  MoveL 5905 to (-69.95, 17.86, -237.76) mm, rotated rx -9.61 ry -16.54 rz -54.03 deg; joints [-14.429, -59.988, 109.983, 192.875, 34.389, -113.768, -415]
  MoveL 5906 to (-68.96, 18.06, -237.77) mm, rotated rx -9.61 ry -16.54 rz -54.03 deg; joints [-14.434, -59.99, 110.053, 192.844, 34.456, -113.734, -415]
  MoveL 5907 to (-67.92, 18.24, -237.77) mm, rotated rx -9.61 ry -16.54 rz -54.03 deg; joints [-14.44, -59.993, 110.127, 192.812, 34.524, -113.701, -415]
  MoveL 5908 to (-67.43, 18.33, -237.77) mm, rotated rx -9.61 ry -16.54 rz -54.03 deg; joints [-14.443, -59.994, 110.162, 192.796, 34.557, -113.684, -415]
  MoveL 5909 to (-66.78, 18.46, -237.8) mm, rotated rx -9.61 ry -16.54 rz -54.03 deg; joints [-14.447, -59.995, 110.208, 192.774, 34.6, -113.662, -415]
  MoveL 5910 to (-66.2, 18.59, -237.86) mm, rotated rx -9.61 ry -16.54 rz -54.03 deg; joints [-14.452, -59.994, 110.248, 192.753, 34.639, -113.64, -415]
  MoveL 5911 to (-65.71, 18.72, -237.93) mm, rotated rx -9.61 ry -16.54 rz -54.03 deg; joints [-14.457, -59.992, 110.28, 192.733, 34.671, -113.622, -415]
  MoveL 5912 to (-65.26, 18.83, -237.99) mm, rotated rx -9.61 ry -16.54 rz -54.03 deg; joints [-14.462, -59.99, 110.31, 192.716, 34.701, -113.605, -415]
  MoveL 5913 to (-64.81, 18.93, -238.02) mm, rotated rx -9.61 ry -16.54 rz -54.03 deg; joints [-14.465, -59.99, 110.341, 192.7, 34.732, -113.589, -415]
  MoveL 5914 to (-63.26, 19.2, -238.02) mm, rotated rx -9.61 ry -16.54 rz -54.03 deg; joints [-14.473, -59.994, 110.452, 192.653, 34.834, -113.539, -415]
  MoveL 5915 to (-62.77, 19.31, -238.03) mm, rotated rx -9.61 ry -16.54 rz -54.03 deg; joints [-14.476, -59.994, 110.486, 192.637, 34.867, -113.522, -415]
  MoveL 5916 to (-62.35, 19.42, -238.06) mm, rotated rx -9.61 ry -16.54 rz -54.03 deg; joints [-14.479, -59.992, 110.514, 192.622, 34.896, -113.507, -415]
  MoveL 5917 to (-61.98, 19.56, -238.11) mm, rotated rx -9.61 ry -16.54 rz -54.03 deg; joints [-14.483, -59.988, 110.537, 192.608, 34.922, -113.494, -415]
  MoveL 5918 to (-61.72, 19.71, -238.17) mm, rotated rx -9.61 ry -16.54 rz -54.03 deg; joints [-14.486, -59.981, 110.549, 192.596, 34.941, -113.482, -415]
  MoveL 5919 to (-61.52, 19.89, -238.24) mm, rotated rx -9.61 ry -16.54 rz -54.03 deg; joints [-14.49, -59.971, 110.558, 192.585, 34.958, -113.472, -415]
  MoveL 5920 to (-63.02, 19.39, -239.05) mm, rotated rx -9.61 ry -16.54 rz -54.03 deg; joints [-14.515, -59.976, 110.447, 192.579, 34.842, -113.488, -415]
  MoveL 5921 to (-61.72, 20.58, -239.45) mm, rotated rx -9.61 ry -16.54 rz -54.03 deg; joints [-14.534, -59.912, 110.497, 192.512, 34.95, -113.424, -415]
  MoveL 5922 to (-60.36, 21.87, -239.71) mm, rotated rx -9.61 ry -16.54 rz -54.03 deg; joints [-14.548, -59.843, 110.549, 192.452, 35.066, -113.364, -415]
  MoveL 5923 to (-58.92, 23.27, -239.9) mm, rotated rx -9.61 ry -16.54 rz -54.03 deg; joints [-14.558, -59.769, 110.603, 192.396, 35.191, -113.305, -415]
  MoveL 5924 to (-57.4, 24.77, -240.09) mm, rotated rx -9.61 ry -16.54 rz -54.03 deg; joints [-14.569, -59.688, 110.659, 192.336, 35.323, -113.243, -415]
  MoveL 5925 to (-55.87, 26.25, -240.18) mm, rotated rx -9.61 ry -16.54 rz -54.03 deg; joints [-14.576, -59.609, 110.718, 192.283, 35.457, -113.184, -415]
  MoveL 5926 to (-54.34, 27.74, -240.28) mm, rotated rx -9.61 ry -16.54 rz -54.03 deg; joints [-14.583, -59.529, 110.777, 192.231, 35.591, -113.126, -415]
  MoveL 5927 to (-52.81, 29.23, -240.48) mm, rotated rx -9.61 ry -16.54 rz -54.03 deg; joints [-14.594, -59.448, 110.833, 192.172, 35.723, -113.065, -415]
  MoveL 5928 to (-51.28, 30.71, -240.58) mm, rotated rx -9.61 ry -16.54 rz -54.03 deg; joints [-14.601, -59.369, 110.891, 192.12, 35.858, -113.008, -415]
  MoveL 5929 to (-49.74, 32.19, -240.68) mm, rotated rx -9.61 ry -16.54 rz -54.03 deg; joints [-14.609, -59.289, 110.949, 192.068, 35.991, -112.951, -415]
  MoveL 5930 to (-48.2, 33.67, -240.88) mm, rotated rx -9.61 ry -16.54 rz -54.03 deg; joints [-14.62, -59.207, 111.005, 192.011, 36.124, -112.891, -415]
  MoveL 5931 to (-45.12, 36.63, -241.08) mm, rotated rx -9.61 ry -16.54 rz -54.03 deg; joints [-14.635, -59.046, 111.12, 191.909, 36.392, -112.779, -415]
  MoveL 5932 to (-43.83, 37.86, -241.29) mm, rotated rx -9.61 ry -16.54 rz -54.03 deg; joints [-14.646, -58.978, 111.167, 191.859, 36.504, -112.728, -415]
  MoveL 5933 to (-42.44, 39.25, -241.36) mm, rotated rx -9.61 ry -16.54 rz -54.03 deg; joints [-14.652, -58.901, 111.216, 191.815, 36.626, -112.679, -415]
  MoveL 5934 to (-41.02, 40.74, -241.37) mm, rotated rx -9.61 ry -16.54 rz -54.03 deg; joints [-14.655, -58.818, 111.264, 191.775, 36.754, -112.631, -415]
  MoveL 5935 to (-39.08, 42.58, -241.48) mm, rotated rx -9.61 ry -16.54 rz -54.03 deg; joints [-14.663, -58.717, 111.335, 191.714, 36.922, -112.563, -415]
  MoveL 5936 to (-37.13, 44.27, -241.58) mm, rotated rx -9.61 ry -16.54 rz -54.03 deg; joints [-14.672, -58.625, 111.413, 191.655, 37.087, -112.498, -415]
  MoveL 5937 to (-35.51, 45.76, -241.67) mm, rotated rx -9.61 ry -16.54 rz -54.03 deg; joints [-14.68, -58.542, 111.475, 191.604, 37.227, -112.442, -415]
  MoveL 5938 to (-34.01, 47.16, -241.84) mm, rotated rx -9.61 ry -16.54 rz -54.03 deg; joints [-14.69, -58.464, 111.528, 191.553, 37.355, -112.389, -415]
  MoveL 5939 to (-32.61, 48.45, -242.13) mm, rotated rx -9.61 ry -16.54 rz -54.03 deg; joints [-14.704, -58.39, 111.577, 191.498, 37.473, -112.334, -415]
  MoveL 5940 to (-31.22, 49.73, -242.41) mm, rotated rx -9.61 ry -16.54 rz -54.03 deg; joints [-14.719, -58.316, 111.625, 191.444, 37.591, -112.28, -415]
  MoveL 5941 to (-29.81, 50.98, -242.71) mm, rotated rx -9.61 ry -16.54 rz -54.03 deg; joints [-14.734, -58.245, 111.675, 191.389, 37.708, -112.226, -415]
  MoveL 5942 to (-28.34, 52.33, -242.86) mm, rotated rx -9.61 ry -16.54 rz -54.03 deg; joints [-14.744, -58.169, 111.728, 191.341, 37.833, -112.176, -415]
  MoveL 5943 to (-27.69, 52.32, -243.48) mm, rotated rx -9.61 ry -16.54 rz -54.03 deg; joints [-14.773, -58.171, 111.768, 191.286, 37.867, -112.136, -415]
  MoveL 5944 to (-27.8, 52.02, -243.79) mm, rotated rx -9.61 ry -16.54 rz -54.03 deg; joints [-14.786, -58.188, 111.767, 191.271, 37.849, -112.129, -415]
  MoveL 5945 to (-27.77, 51.98, -243.98) mm, rotated rx -9.61 ry -16.54 rz -54.03 deg; joints [-14.794, -58.189, 111.768, 191.258, 37.847, -112.122, -415]
  MoveL 5946 to (-27.63, 52.19, -244.08) mm, rotated rx -9.61 ry -16.54 rz -54.03 deg; joints [-14.798, -58.176, 111.768, 191.249, 37.86, -112.114, -415]
  MoveL 5947 to (-27.45, 52.6, -244.1) mm, rotated rx -9.61 ry -16.54 rz -54.03 deg; joints [-14.798, -58.15, 111.764, 191.243, 37.882, -112.107, -415]
  MoveL 5948 to (-27.29, 53.06, -244.1) mm, rotated rx -9.61 ry -16.54 rz -54.03 deg; joints [-14.798, -58.12, 111.757, 191.238, 37.904, -112.1, -415]
  MoveL 5949 to (-27.08, 54.01, -244.14) mm, rotated rx -9.61 ry -16.54 rz -54.03 deg; joints [-14.796, -58.058, 111.733, 191.231, 37.941, -112.089, -415]
  MoveL 5950 to (-26.74, 55.55, -244.14) mm, rotated rx -9.61 ry -16.54 rz -54.03 deg; joints [-14.792, -57.958, 111.694, 191.222, 38.002, -112.074, -415]
  MoveL 5951 to (-26.49, 56.5, -244.15) mm, rotated rx -9.61 ry -16.54 rz -54.03 deg; joints [-14.79, -57.896, 111.672, 191.215, 38.041, -112.063, -415]
  MoveL 5952 to (-26.27, 57.52, -244.15) mm, rotated rx -9.61 ry -16.54 rz -54.03 deg; joints [-14.788, -57.829, 111.646, 191.209, 38.081, -112.053, -415]
  MoveL 5953 to (-26.15, 58.02, -244.17) mm, rotated rx -9.61 ry -16.54 rz -54.03 deg; joints [-14.787, -57.796, 111.633, 191.205, 38.101, -112.047, -415]
  MoveL 5954 to (-26.04, 58.48, -244.2) mm, rotated rx -9.61 ry -16.54 rz -54.03 deg; joints [-14.787, -57.767, 111.622, 191.2, 38.12, -112.041, -415]
  MoveL 5955 to (-25.92, 58.9, -244.24) mm, rotated rx -9.61 ry -16.54 rz -54.03 deg; joints [-14.788, -57.739, 111.612, 191.194, 38.137, -112.035, -415]
  MoveL 5956 to (-25.81, 59.29, -244.31) mm, rotated rx -9.61 ry -16.54 rz -54.03 deg; joints [-14.789, -57.713, 111.604, 191.188, 38.153, -112.028, -415]
  MoveL 5957 to (-25.69, 59.69, -244.36) mm, rotated rx -9.61 ry -16.54 rz -54.03 deg; joints [-14.791, -57.687, 111.595, 191.182, 38.17, -112.021, -415]
  MoveL 5958 to (-25.57, 60.14, -244.39) mm, rotated rx -9.61 ry -16.54 rz -54.03 deg; joints [-14.791, -57.658, 111.584, 191.177, 38.188, -112.015, -415]
  MoveL 5959 to (-25.46, 60.6, -244.42) mm, rotated rx -9.61 ry -16.54 rz -54.03 deg; joints [-14.791, -57.627, 111.573, 191.172, 38.207, -112.009, -415]
  MoveL 5960 to (-25.34, 61.02, -244.46) mm, rotated rx -9.61 ry -16.54 rz -54.03 deg; joints [-14.792, -57.6, 111.563, 191.167, 38.225, -112.003, -415]
  MoveL 5961 to (-25.21, 61.41, -244.52) mm, rotated rx -9.61 ry -16.54 rz -54.03 deg; joints [-14.793, -57.575, 111.556, 191.16, 38.242, -111.996, -415]
  MoveL 5962 to (-25.09, 61.8, -244.57) mm, rotated rx -9.61 ry -16.54 rz -54.03 deg; joints [-14.794, -57.549, 111.547, 191.154, 38.259, -111.99, -415]
  MoveL 5963 to (-24.97, 62.22, -244.6) mm, rotated rx -9.61 ry -16.54 rz -54.03 deg; joints [-14.795, -57.521, 111.537, 191.149, 38.276, -111.984, -415]
  MoveL 5964 to (-24.86, 62.73, -244.6) mm, rotated rx -9.61 ry -16.54 rz -54.03 deg; joints [-14.793, -57.488, 111.524, 191.146, 38.296, -111.979, -415]
  MoveL 5965 to (-23.99, 65.52, -244.96) mm, rotated rx -9.61 ry -16.54 rz -54.03 deg; joints [-14.802, -57.306, 111.465, 191.103, 38.416, -111.933, -415]
  MoveL 5966 to (-23.41, 66.67, -245.4) mm, rotated rx -9.61 ry -16.54 rz -54.03 deg; joints [-14.818, -57.23, 111.452, 191.063, 38.476, -111.898, -415]
  MoveL 5967 to (-22.74, 67.66, -246.03) mm, rotated rx -9.61 ry -16.54 rz -54.03 deg; joints [-14.843, -57.164, 111.451, 191.009, 38.536, -111.855, -415]
  MoveL 5968 to (-21.11, 69.17, -247.81) mm, rotated rx -9.61 ry -16.54 rz -54.03 deg; joints [-14.918, -57.064, 111.48, 190.863, 38.655, -111.747, -415]
  MoveL 5969 to (-19.1, 70.04, -250.3) mm, rotated rx -9.61 ry -16.54 rz -54.03 deg; joints [-15.027, -57.003, 111.553, 190.666, 38.775, -111.607, -415]
  MoveL 5970 to (-17.3, 70.14, -252.79) mm, rotated rx -9.61 ry -16.54 rz -54.03 deg; joints [-15.138, -56.991, 111.643, 190.475, 38.863, -111.477, -415]
  MoveL 5971 to (-16.71, 69.87, -253.77) mm, rotated rx -9.61 ry -16.54 rz -54.03 deg; joints [-15.182, -57.008, 111.684, 190.402, 38.882, -111.43, -415]
  MoveL 5972 to (-16.31, 69.36, -254.58) mm, rotated rx -9.61 ry -16.54 rz -54.03 deg; joints [-15.218, -57.038, 111.722, 190.345, 38.886, -111.395, -415]
  MoveL 5973 to (-16.19, 69.03, -254.91) mm, rotated rx -9.61 ry -16.54 rz -54.03 deg; joints [-15.234, -57.059, 111.74, 190.321, 38.881, -111.382, -415]
  MoveL 5974 to (-16.12, 68.64, -255.2) mm, rotated rx -9.61 ry -16.54 rz -54.03 deg; joints [-15.248, -57.084, 111.757, 190.302, 38.873, -111.371, -415]
  MoveL 5975 to (-16.13, 67.69, -255.64) mm, rotated rx -9.61 ry -16.54 rz -54.03 deg; joints [-15.269, -57.144, 111.79, 190.275, 38.844, -111.359, -415]
  MoveL 5976 to (-16.34, 66.52, -255.91) mm, rotated rx -9.61 ry -16.54 rz -54.03 deg; joints [-15.284, -57.219, 111.82, 190.263, 38.798, -111.359, -415]
  MoveL 5977 to (-16.76, 65.13, -256) mm, rotated rx -9.61 ry -16.54 rz -54.03 deg; joints [-15.291, -57.308, 111.847, 190.267, 38.736, -111.37, -415]
  MoveL 5978 to (-17.61, 62.66, -256) mm, rotated rx -9.61 ry -16.54 rz -54.03 deg; joints [-15.296, -57.468, 111.89, 190.285, 38.621, -111.399, -415]
  MoveL 5979 to (-17.76, 62.25, -255.97) mm, rotated rx -9.61 ry -16.54 rz -54.03 deg; joints [-15.295, -57.494, 111.896, 190.29, 38.601, -111.405, -415]
  MoveL 5980 to (-17.92, 61.87, -255.92) mm, rotated rx -9.61 ry -16.54 rz -54.03 deg; joints [-15.294, -57.518, 111.901, 190.296, 38.582, -111.412, -415]
  MoveL 5981 to (-18.08, 61.52, -255.85) mm, rotated rx -9.61 ry -16.54 rz -54.03 deg; joints [-15.292, -57.541, 111.906, 190.304, 38.564, -111.42, -415]
  MoveL 5982 to (-18.24, 61.12, -255.8) mm, rotated rx -9.61 ry -16.54 rz -54.03 deg; joints [-15.29, -57.567, 111.911, 190.311, 38.544, -111.427, -415]
  MoveL 5983 to (-18.42, 60.66, -255.76) mm, rotated rx -9.61 ry -16.54 rz -54.03 deg; joints [-15.29, -57.597, 111.918, 190.317, 38.522, -111.434, -415]
  MoveL 5984 to (-18.62, 60.17, -255.71) mm, rotated rx -9.61 ry -16.54 rz -54.03 deg; joints [-15.288, -57.629, 111.925, 190.325, 38.497, -111.442, -415]
  MoveL 5985 to (-18.81, 59.66, -255.69) mm, rotated rx -9.61 ry -16.54 rz -54.03 deg; joints [-15.288, -57.661, 111.933, 190.33, 38.473, -111.449, -415]
  MoveL 5986 to (-19.01, 59.05, -255.7) mm, rotated rx -9.61 ry -16.54 rz -54.03 deg; joints [-15.29, -57.7, 111.943, 190.333, 38.444, -111.456, -415]
  MoveL 5987 to (-19.27, 58.22, -255.77) mm, rotated rx -9.61 ry -16.54 rz -54.03 deg; joints [-15.295, -57.754, 111.958, 190.335, 38.406, -111.463, -415]
  MoveL 5988 to (-19.44, 57.72, -255.77) mm, rotated rx -9.61 ry -16.54 rz -54.03 deg; joints [-15.296, -57.785, 111.966, 190.339, 38.383, -111.468, -415]
  MoveL 5989 to (-19.6, 57.25, -255.76) mm, rotated rx -9.61 ry -16.54 rz -54.03 deg; joints [-15.297, -57.816, 111.974, 190.343, 38.361, -111.474, -415]
  MoveL 5990 to (-19.76, 56.82, -255.74) mm, rotated rx -9.61 ry -16.54 rz -54.03 deg; joints [-15.297, -57.844, 111.981, 190.348, 38.34, -111.481, -415]
  MoveL 5991 to (-19.92, 56.43, -255.69) mm, rotated rx -9.61 ry -16.54 rz -54.03 deg; joints [-15.295, -57.869, 111.985, 190.354, 38.32, -111.488, -415]
  MoveL 5992 to (-20.09, 56.07, -255.63) mm, rotated rx -9.61 ry -16.54 rz -54.03 deg; joints [-15.293, -57.892, 111.989, 190.362, 38.301, -111.495, -415]
  MoveL 5993 to (-20.31, 55.71, -255.58) mm, rotated rx -9.61 ry -16.54 rz -54.03 deg; joints [-15.291, -57.914, 111.988, 190.37, 38.279, -111.504, -415]
  MoveL 5994 to (-20.56, 55.39, -255.52) mm, rotated rx -9.61 ry -16.54 rz -54.03 deg; joints [-15.289, -57.935, 111.984, 190.379, 38.255, -111.513, -415]
  MoveL 5995 to (-20.74, 55.25, -255.36) mm, rotated rx -9.61 ry -16.54 rz -54.03 deg; joints [-15.282, -57.943, 111.979, 190.394, 38.242, -111.524, -415]
  MoveL 5996 to (-20.74, 55.36, -255.05) mm, rotated rx -9.61 ry -16.54 rz -54.03 deg; joints [-15.269, -57.939, 111.979, 190.413, 38.248, -111.534, -415]
  MoveL 5997 to (-20.54, 55.75, -254.56) mm, rotated rx -9.61 ry -16.54 rz -54.03 deg; joints [-15.249, -57.919, 111.987, 190.437, 38.277, -111.545, -415]
  MoveL 5998 to (-21.22, 55.18, -253.71) mm, rotated rx -9.61 ry -16.54 rz -54.03 deg; joints [-15.212, -57.957, 111.973, 190.505, 38.229, -111.594, -415]
  MoveL 5999 to (-24.62, 52.6, -253.71) mm, rotated rx -9.61 ry -16.54 rz -54.03 deg; joints [-15.202, -58.097, 111.825, 190.589, 37.948, -111.689, -415]
  MoveL 6000 to (-26.22, 51.39, -253.64) mm, rotated rx -9.61 ry -16.54 rz -54.03 deg; joints [-15.194, -58.162, 111.756, 190.632, 37.817, -111.737, -415]
  MoveL 6001 to (-27.81, 50.2, -253.49) mm, rotated rx -9.61 ry -16.54 rz -54.03 deg; joints [-15.183, -58.227, 111.688, 190.681, 37.687, -111.788, -415]
  MoveL 6002 to (-29.65, 48.83, -253.3) mm, rotated rx -9.61 ry -16.54 rz -54.03 deg; joints [-15.17, -58.301, 111.609, 190.739, 37.538, -111.847, -415]
  MoveL 6003 to (-31.39, 47.53, -253.08) mm, rotated rx -9.61 ry -16.54 rz -54.03 deg; joints [-15.156, -58.371, 111.534, 190.797, 37.397, -111.905, -415]
  MoveL 6004 to (-33.13, 46.22, -252.98) mm, rotated rx -9.61 ry -16.54 rz -54.03 deg; joints [-15.146, -58.441, 111.458, 190.848, 37.255, -111.96, -415]
  MoveL 6005 to (-34.83, 44.93, -252.98) mm, rotated rx -9.61 ry -16.54 rz -54.03 deg; joints [-15.141, -58.509, 111.382, 190.892, 37.114, -112.01, -415]
  MoveL 6006 to (-36.41, 43.72, -252.92) mm, rotated rx -9.61 ry -16.54 rz -54.03 deg; joints [-15.134, -58.572, 111.312, 190.937, 36.984, -112.059, -415]
  MoveL 6007 to (-37.9, 42.58, -252.8) mm, rotated rx -9.61 ry -16.54 rz -54.03 deg; joints [-15.124, -58.633, 111.247, 190.983, 36.862, -112.108, -415]
  MoveL 6008 to (-39.53, 41.35, -252.73) mm, rotated rx -9.61 ry -16.54 rz -54.03 deg; joints [-15.117, -58.697, 111.174, 191.03, 36.729, -112.159, -415]
  MoveL 6009 to (-41.22, 40.05, -252.55) mm, rotated rx -9.61 ry -16.54 rz -54.03 deg; joints [-15.104, -58.765, 111.1, 191.087, 36.591, -112.217, -415]
  MoveL 6010 to (-44.62, 37.46, -252.37) mm, rotated rx -9.61 ry -16.54 rz -54.03 deg; joints [-15.087, -58.899, 110.948, 191.19, 36.312, -112.328, -415]
  MoveL 6011 to (-46.31, 36.16, -252.19) mm, rotated rx -9.61 ry -16.54 rz -54.03 deg; joints [-15.074, -58.967, 110.873, 191.247, 36.174, -112.387, -415]
  MoveL 6012 to (-48, 34.85, -252.01) mm, rotated rx -9.61 ry -16.54 rz -54.03 deg; joints [-15.062, -59.034, 110.799, 191.305, 36.036, -112.447, -415]
  MoveL 6013 to (-49.7, 33.56, -252.01) mm, rotated rx -9.61 ry -16.54 rz -54.03 deg; joints [-15.057, -59.099, 110.72, 191.352, 35.896, -112.501, -415]
  MoveL 6014 to (-51.38, 32.25, -251.83) mm, rotated rx -9.61 ry -16.54 rz -54.03 deg; joints [-15.045, -59.166, 110.645, 191.411, 35.758, -112.561, -415]
  MoveL 6015 to (-53.06, 30.94, -251.66) mm, rotated rx -9.61 ry -16.54 rz -54.03 deg; joints [-15.033, -59.233, 110.57, 191.47, 35.62, -112.622, -415]
  MoveL 6016 to (-54.76, 29.65, -251.66) mm, rotated rx -9.61 ry -16.54 rz -54.03 deg; joints [-15.028, -59.297, 110.49, 191.518, 35.48, -112.677, -415]
  MoveL 6017 to (-56.27, 28.41, -251.46) mm, rotated rx -9.61 ry -16.54 rz -54.03 deg; joints [-15.016, -59.361, 110.425, 191.574, 35.355, -112.734, -415]
  MoveL 6018 to (-57.55, 27.27, -251.14) mm, rotated rx -9.61 ry -16.54 rz -54.03 deg; joints [-15, -59.422, 110.376, 191.632, 35.249, -112.789, -415]
  MoveL 6019 to (-58.64, 26.2, -250.68) mm, rotated rx -9.61 ry -16.54 rz -54.03 deg; joints [-14.979, -59.483, 110.341, 191.693, 35.158, -112.845, -415]
  MoveL 6020 to (-57.79, 26.63, -249.91) mm, rotated rx -9.61 ry -16.54 rz -54.03 deg; joints [-14.952, -59.473, 110.402, 191.718, 35.231, -112.849, -415]
  MoveL 6021 to (-58.15, 26.41, -249.9) mm, rotated rx -9.61 ry -16.54 rz -54.03 deg; joints [-14.95, -59.482, 110.383, 191.729, 35.204, -112.861, -415]
  MoveC 6022 to (-61.66, 25.91, -249.9) mm, rotated rx -9.61 ry -16.54 rz -54.03 deg; joints [-14.931, -59.467, 110.129, 191.83, 34.972, -112.967, -415] to (-65.21, 25.71, -249.9) mm, rotated rx -9.61 ry -16.54 rz -54.03 deg; joints [-14.91, -59.43, 109.859, 191.934, 34.747, -113.073, -415]
  MoveL 6023 to (-65.21, 25.71, -249.9) mm, rotated rx -9.61 ry -16.54 rz -54.03 deg; joints [-14.91, -59.43, 109.859, 191.934, 34.747, -113.073, -415]
  MoveL 6024 to (-65.68, 25.67, -249.88) mm, rotated rx -9.61 ry -16.54 rz -54.03 deg; joints [-14.907, -59.426, 109.825, 191.949, 34.717, -113.088, -415]
  MoveL 6025 to (-66.1, 25.62, -249.83) mm, rotated rx -9.61 ry -16.54 rz -54.03 deg; joints [-14.902, -59.425, 109.795, 191.964, 34.691, -113.103, -415]
  MoveL 6026 to (-66.5, 25.56, -249.77) mm, rotated rx -9.61 ry -16.54 rz -54.03 deg; joints [-14.898, -59.423, 109.767, 191.98, 34.665, -113.118, -415]
  MoveL 6027 to (-66.94, 25.51, -249.72) mm, rotated rx -9.61 ry -16.54 rz -54.03 deg; joints [-14.893, -59.421, 109.735, 191.996, 34.637, -113.133, -415]
  MoveL 6028 to (-67.41, 25.46, -249.7) mm, rotated rx -9.61 ry -16.54 rz -54.03 deg; joints [-14.89, -59.417, 109.7, 192.012, 34.607, -113.149, -415]
  MoveL 6029 to (-67.93, 25.43, -249.68) mm, rotated rx -9.61 ry -16.54 rz -54.03 deg; joints [-14.886, -59.412, 109.662, 192.028, 34.575, -113.165, -415]
  MoveL 6030 to (-68.97, 25.36, -249.68) mm, rotated rx -9.61 ry -16.54 rz -54.03 deg; joints [-14.88, -59.401, 109.582, 192.059, 34.508, -113.197, -415]
  MoveL 6031 to (-70.43, 25.33, -249.77) mm, rotated rx -9.61 ry -16.54 rz -54.03 deg; joints [-14.875, -59.381, 109.467, 192.096, 34.416, -113.238, -415]
  MoveL 6032 to (-71.62, 25.43, -250.05) mm, rotated rx -9.61 ry -16.54 rz -54.03 deg; joints [-14.878, -59.355, 109.365, 192.114, 34.342, -113.262, -415]
  MoveL 6033 to (-72.56, 25.67, -250.5) mm, rotated rx -9.61 ry -16.54 rz -54.03 deg; joints [-14.89, -59.322, 109.275, 192.112, 34.285, -113.271, -415]
  MoveL 6034 to (-73.24, 26.03, -251.14) mm, rotated rx -9.61 ry -16.54 rz -54.03 deg; joints [-14.91, -59.282, 109.197, 192.09, 34.244, -113.263, -415]
  MoveL 6035 to (-73.67, 26.52, -251.97) mm, rotated rx -9.61 ry -16.54 rz -54.03 deg; joints [-14.938, -59.236, 109.131, 192.049, 34.221, -113.239, -415]
  MoveL 6036 to (-73.83, 27.14, -252.97) mm, rotated rx -9.61 ry -16.54 rz -54.03 deg; joints [-14.974, -59.183, 109.077, 191.988, 34.215, -113.198, -415]
  MoveL 6037 to (-73.39, 28.77, -255.53) mm, rotated rx -9.61 ry -16.54 rz -54.03 deg; joints [-15.071, -59.059, 109.007, 191.807, 34.255, -113.07, -415]
  MoveL 6038 to (-72.15, 30.4, -258.09) mm, rotated rx -9.61 ry -16.54 rz -54.03 deg; joints [-15.173, -58.946, 108.997, 191.604, 34.343, -112.918, -415]
  MoveL 6039 to (-71.32, 31.03, -259.1) mm, rotated rx -9.61 ry -16.54 rz -54.03 deg; joints [-15.215, -58.907, 109.021, 191.515, 34.399, -112.849, -415]
  MoveL 6040 to (-70.36, 31.53, -259.92) mm, rotated rx -9.61 ry -16.54 rz -54.03 deg; joints [-15.252, -58.881, 109.063, 191.434, 34.462, -112.785, -415]
  MoveL 6041 to (-69.26, 31.9, -260.56) mm, rotated rx -9.61 ry -16.54 rz -54.03 deg; joints [-15.282, -58.866, 109.124, 191.36, 34.532, -112.724, -415]
  MoveL 6042 to (-68.01, 32.14, -261.02) mm, rotated rx -9.61 ry -16.54 rz -54.03 deg; joints [-15.307, -58.864, 109.204, 191.295, 34.61, -112.669, -415]
  MoveL 6043 to (-65.12, 32.24, -261.38) mm, rotated rx -9.61 ry -16.54 rz -54.03 deg; joints [-15.339, -58.894, 109.421, 191.189, 34.788, -112.57, -415]
  MoveL 6044 to (-64.07, 32.19, -261.38) mm, rotated rx -9.61 ry -16.54 rz -54.03 deg; joints [-15.346, -58.912, 109.505, 191.159, 34.852, -112.54, -415]
  MoveL 6045 to (-63.55, 32.17, -261.39) mm, rotated rx -9.61 ry -16.54 rz -54.03 deg; joints [-15.35, -58.921, 109.546, 191.144, 34.884, -112.525, -415]
  MoveL 6046 to (-63.07, 32.16, -261.41) mm, rotated rx -9.61 ry -16.54 rz -54.03 deg; joints [-15.354, -58.928, 109.583, 191.129, 34.913, -112.51, -415]
  MoveL 6047 to (-62.65, 32.17, -261.46) mm, rotated rx -9.61 ry -16.54 rz -54.03 deg; joints [-15.358, -58.933, 109.616, 191.114, 34.939, -112.496, -415]
  MoveL 6048 to (-62.25, 32.18, -261.52) mm, rotated rx -9.61 ry -16.54 rz -54.03 deg; joints [-15.363, -58.937, 109.646, 191.099, 34.963, -112.483, -415]
  MoveL 6049 to (-61.83, 32.18, -261.56) mm, rotated rx -9.61 ry -16.54 rz -54.03 deg; joints [-15.367, -58.942, 109.677, 191.084, 34.989, -112.469, -415]
  MoveL 6050 to (-61.36, 32.17, -261.59) mm, rotated rx -9.61 ry -16.54 rz -54.03 deg; joints [-15.371, -58.949, 109.714, 191.07, 35.018, -112.455, -415]
  MoveL 6051 to (-60.86, 32.15, -261.59) mm, rotated rx -9.61 ry -16.54 rz -54.03 deg; joints [-15.375, -58.957, 109.753, 191.056, 35.048, -112.44, -415]
  MoveL 6052 to (-60.31, 32.12, -261.59) mm, rotated rx -9.61 ry -16.54 rz -54.03 deg; joints [-15.378, -58.967, 109.798, 191.041, 35.082, -112.425, -415]
  MoveL 6053 to (-59.78, 32.1, -261.59) mm, rotated rx -9.61 ry -16.54 rz -54.03 deg; joints [-15.382, -58.976, 109.84, 191.025, 35.114, -112.41, -415]
  MoveL 6054 to (-59.29, 32.09, -261.62) mm, rotated rx -9.61 ry -16.54 rz -54.03 deg; joints [-15.386, -58.983, 109.878, 191.01, 35.144, -112.395, -415]
  MoveL 6055 to (-58.81, 32.08, -261.66) mm, rotated rx -9.61 ry -16.54 rz -54.03 deg; joints [-15.391, -58.989, 109.914, 190.994, 35.173, -112.38, -415]
  MoveL 6056 to (-58.31, 32.1, -261.74) mm, rotated rx -9.61 ry -16.54 rz -54.03 deg; joints [-15.397, -58.995, 109.952, 190.975, 35.204, -112.363, -415]
  MoveL 6057 to (-57.7, 32.11, -261.8) mm, rotated rx -9.61 ry -16.54 rz -54.03 deg; joints [-15.403, -59.002, 109.997, 190.954, 35.241, -112.343, -415]
  MoveL 6058 to (-57.13, 32.09, -261.82) mm, rotated rx -9.61 ry -16.54 rz -54.03 deg; joints [-15.408, -59.01, 110.042, 190.937, 35.276, -112.327, -415]
  MoveL 6059 to (-56.61, 32.07, -261.82) mm, rotated rx -9.61 ry -16.54 rz -54.03 deg; joints [-15.411, -59.019, 110.084, 190.922, 35.308, -112.312, -415]
  MoveL 6060 to (-56.08, 32.04, -261.82) mm, rotated rx -9.61 ry -16.54 rz -54.03 deg; joints [-15.415, -59.027, 110.125, 190.908, 35.34, -112.298, -415]
  MoveL 6061 to (-55.42, 32.03, -261.83) mm, rotated rx -9.61 ry -16.54 rz -54.03 deg; joints [-15.419, -59.037, 110.177, 190.889, 35.381, -112.279, -415]
  MoveL 6062 to (-54.84, 32.04, -261.84) mm, rotated rx -9.61 ry -16.54 rz -54.03 deg; joints [-15.423, -59.044, 110.222, 190.873, 35.417, -112.262, -415]
  MoveL 6063 to (-54.33, 32.07, -261.85) mm, rotated rx -9.61 ry -16.54 rz -54.03 deg; joints [-15.427, -59.048, 110.259, 190.858, 35.449, -112.248, -415]
  MoveL 6064 to (-54, 32.15, -261.85) mm, rotated rx -9.61 ry -16.54 rz -54.03 deg; joints [-15.429, -59.048, 110.282, 190.849, 35.472, -112.238, -415]
  MoveL 6065 to (-53.75, 32.25, -261.85) mm, rotated rx -9.61 ry -16.54 rz -54.03 deg; joints [-15.43, -59.044, 110.298, 190.842, 35.491, -112.231, -415]
  MoveL 6066 to (-54.61, 31.88, -262.44) mm, rotated rx -9.61 ry -16.54 rz -54.03 deg; joints [-15.449, -59.052, 110.235, 190.828, 35.42, -112.233, -415]
  MoveL 6067 to (-53.63, 32.79, -262.97) mm, rotated rx -9.61 ry -16.54 rz -54.03 deg; joints [-15.473, -58.999, 110.266, 190.768, 35.499, -112.181, -415]
  MoveL 6068 to (-52.4, 33.75, -263.35) mm, rotated rx -9.61 ry -16.54 rz -54.03 deg; joints [-15.492, -58.948, 110.317, 190.71, 35.597, -112.128, -415]
  MoveL 6069 to (-50.87, 34.78, -263.61) mm, rotated rx -9.61 ry -16.54 rz -54.03 deg; joints [-15.507, -58.897, 110.389, 190.653, 35.716, -112.073, -415]
  MoveL 6070 to (-49.13, 35.87, -263.74) mm, rotated rx -9.61 ry -16.54 rz -54.03 deg; joints [-15.519, -58.846, 110.478, 190.598, 35.853, -112.017, -415]
  MoveL 6071 to (-47.33, 36.97, -263.83) mm, rotated rx -9.61 ry -16.54 rz -54.03 deg; joints [-15.529, -58.794, 110.57, 190.545, 35.993, -111.961, -415]
  MoveL 6072 to (-43.69, 39.18, -264.01) mm, rotated rx -9.61 ry -16.54 rz -54.03 deg; joints [-15.55, -58.69, 110.758, 190.438, 36.277, -111.849, -415]
  MoveL 6073 to (-41.87, 40.3, -264.19) mm, rotated rx -9.61 ry -16.54 rz -54.03 deg; joints [-15.564, -58.636, 110.849, 190.38, 36.419, -111.79, -415]
  MoveL 6074 to (-38.22, 42.51, -264.37) mm, rotated rx -9.61 ry -16.54 rz -54.03 deg; joints [-15.586, -58.53, 111.035, 190.275, 36.704, -111.681, -415]
  MoveL 6075 to (-36.39, 43.61, -264.55) mm, rotated rx -9.61 ry -16.54 rz -54.03 deg; joints [-15.6, -58.475, 111.126, 190.218, 36.845, -111.624, -415]
  MoveL 6076 to (-34.56, 44.71, -264.64) mm, rotated rx -9.61 ry -16.54 rz -54.03 deg; joints [-15.611, -58.422, 111.218, 190.166, 36.988, -111.57, -415]
  MoveL 6077 to (-32.86, 45.71, -264.86) mm, rotated rx -9.61 ry -16.54 rz -54.03 deg; joints [-15.626, -58.372, 111.303, 190.111, 37.119, -111.516, -415]
  MoveL 6078 to (-30.84, 46.93, -265) mm, rotated rx -9.61 ry -16.54 rz -54.03 deg; joints [-15.639, -58.311, 111.404, 190.052, 37.276, -111.456, -415]
  MoveL 6079 to (-28.64, 48.25, -265.12) mm, rotated rx -9.61 ry -16.54 rz -54.03 deg; joints [-15.653, -58.245, 111.513, 189.991, 37.447, -111.392, -415]
  MoveL 6080 to (-26.82, 49.35, -265.12) mm, rotated rx -9.61 ry -16.54 rz -54.03 deg; joints [-15.66, -58.191, 111.606, 189.947, 37.591, -111.344, -415]
  MoveL 6081 to (-25.07, 50.39, -265.2) mm, rotated rx -9.61 ry -16.54 rz -54.03 deg; joints [-15.67, -58.139, 111.693, 189.9, 37.728, -111.295, -415]
  MoveL 6082 to (-23.49, 51.32, -265.37) mm, rotated rx -9.61 ry -16.54 rz -54.03 deg; joints [-15.683, -58.091, 111.771, 189.852, 37.85, -111.247, -415]
  MoveL 6083 to (-21.87, 52.25, -265.58) mm, rotated rx -9.61 ry -16.54 rz -54.03 deg; joints [-15.698, -58.043, 111.85, 189.801, 37.974, -111.198, -415]
  MoveL 6084 to (-19.84, 53.45, -265.72) mm, rotated rx -9.61 ry -16.54 rz -54.03 deg; joints [-15.711, -57.981, 111.95, 189.745, 38.132, -111.14, -415]
  MoveL 6085 to (-17.63, 54.77, -265.82) mm, rotated rx -9.61 ry -16.54 rz -54.03 deg; joints [-15.724, -57.913, 112.059, 189.687, 38.305, -111.08, -415]
  MoveL 6086 to (-13.97, 56.97, -265.82) mm, rotated rx -9.61 ry -16.54 rz -54.03 deg; joints [-15.739, -57.8, 112.24, 189.603, 38.594, -110.988, -415]
  MoveL 6087 to (-13.67, 56.88, -266.52) mm, rotated rx -9.61 ry -16.54 rz -54.03 deg; joints [-15.769, -57.802, 112.254, 189.554, 38.602, -110.956, -415]
  MoveL 6088 to (-13.85, 56.63, -266.86) mm, rotated rx -9.61 ry -16.54 rz -54.03 deg; joints [-15.783, -57.815, 112.245, 189.537, 38.58, -110.949, -415]
  MoveL 6089 to (-13.84, 56.61, -267.08) mm, rotated rx -9.61 ry -16.54 rz -54.03 deg; joints [-15.792, -57.814, 112.243, 189.524, 38.578, -110.942, -415]
  MoveL 6090 to (-13.67, 56.82, -267.19) mm, rotated rx -9.61 ry -16.54 rz -54.03 deg; joints [-15.796, -57.801, 112.245, 189.513, 38.592, -110.933, -415]
  MoveL 6091 to (-13.43, 57.2, -267.22) mm, rotated rx -9.61 ry -16.54 rz -54.03 deg; joints [-15.798, -57.777, 112.247, 189.506, 38.617, -110.925, -415]
  MoveL 6092 to (-13.19, 57.61, -267.25) mm, rotated rx -9.61 ry -16.54 rz -54.03 deg; joints [-15.798, -57.751, 112.246, 189.5, 38.642, -110.918, -415]
  MoveL 6093 to (-12.99, 57.99, -267.3) mm, rotated rx -9.61 ry -16.54 rz -54.03 deg; joints [-15.8, -57.727, 112.245, 189.493, 38.665, -110.911, -415]
  MoveL 6094 to (-12.79, 58.34, -267.37) mm, rotated rx -9.61 ry -16.54 rz -54.03 deg; joints [-15.802, -57.704, 112.244, 189.485, 38.685, -110.903, -415]
  MoveL 6095 to (-12.59, 58.7, -267.42) mm, rotated rx -9.61 ry -16.54 rz -54.03 deg; joints [-15.804, -57.681, 112.242, 189.477, 38.706, -110.895, -415]
  MoveL 6096 to (-12.38, 59.09, -267.46) mm, rotated rx -9.61 ry -16.54 rz -54.03 deg; joints [-15.806, -57.656, 112.24, 189.471, 38.729, -110.888, -415]
  MoveL 6097 to (-12.15, 59.56, -267.49) mm, rotated rx -9.61 ry -16.54 rz -54.03 deg; joints [-15.806, -57.627, 112.237, 189.464, 38.756, -110.881, -415]
  MoveL 6098 to (-11.9, 60.03, -267.55) mm, rotated rx -9.61 ry -16.54 rz -54.03 deg; joints [-15.808, -57.597, 112.235, 189.455, 38.783, -110.871, -415]
  MoveL 6099 to (-11.66, 60.49, -267.58) mm, rotated rx -9.61 ry -16.54 rz -54.03 deg; joints [-15.809, -57.567, 112.233, 189.449, 38.809, -110.864, -415]
  MoveL 6100 to (-11.44, 60.96, -267.59) mm, rotated rx -9.61 ry -16.54 rz -54.03 deg; joints [-15.809, -57.537, 112.229, 189.444, 38.835, -110.857, -415]
  MoveL 6101 to (-11.22, 61.44, -267.59) mm, rotated rx -9.61 ry -16.54 rz -54.03 deg; joints [-15.808, -57.507, 112.225, 189.44, 38.861, -110.851, -415]
  MoveL 6102 to (-10.94, 62.07, -267.55) mm, rotated rx -9.61 ry -16.54 rz -54.03 deg; joints [-15.806, -57.467, 112.22, 189.436, 38.895, -110.844, -415]
  MoveL 6103 to (-10.67, 62.67, -267.52) mm, rotated rx -9.61 ry -16.54 rz -54.03 deg; joints [-15.803, -57.429, 112.214, 189.433, 38.928, -110.837, -415]
  MoveL 6104 to (-10.42, 63.22, -267.52) mm, rotated rx -9.61 ry -16.54 rz -54.03 deg; joints [-15.802, -57.394, 112.21, 189.428, 38.958, -110.83, -415]
  MoveL 6105 to (-10.2, 63.63, -267.55) mm, rotated rx -9.61 ry -16.54 rz -54.03 deg; joints [-15.803, -57.368, 112.207, 189.422, 38.981, -110.823, -415]
  MoveL 6106 to (-10, 63.99, -267.61) mm, rotated rx -9.61 ry -16.54 rz -54.03 deg; joints [-15.806, -57.345, 112.206, 189.414, 39.003, -110.816, -415]
  MoveL 6107 to (-9.8, 64.35, -267.67) mm, rotated rx -9.61 ry -16.54 rz -54.03 deg; joints [-15.807, -57.322, 112.204, 189.407, 39.024, -110.808, -415]
  MoveL 6108 to (-9.6, 64.74, -267.7) mm, rotated rx -9.61 ry -16.54 rz -54.03 deg; joints [-15.808, -57.297, 112.202, 189.401, 39.046, -110.801, -415]
  MoveL 6109 to (-8.93, 66.17, -267.7) mm, rotated rx -9.61 ry -16.54 rz -54.03 deg; joints [-15.807, -57.206, 112.191, 189.388, 39.124, -110.783, -415]
  MoveL 6110 to (-7.5, 68.68, -268.08) mm, rotated rx -9.61 ry -16.54 rz -54.03 deg; joints [-15.82, -57.045, 112.182, 189.337, 39.273, -110.732, -415]
  MoveL 6111 to (-6.72, 69.66, -268.55) mm, rotated rx -9.61 ry -16.54 rz -54.03 deg; joints [-15.84, -56.981, 112.189, 189.294, 39.341, -110.696, -415]
  MoveL 6112 to (-5.91, 70.46, -269.21) mm, rotated rx -9.61 ry -16.54 rz -54.03 deg; joints [-15.868, -56.927, 112.203, 189.238, 39.406, -110.654, -415]
  MoveL 6113 to (-5.05, 71.09, -270.06) mm, rotated rx -9.61 ry -16.54 rz -54.03 deg; joints [-15.905, -56.885, 112.225, 189.17, 39.466, -110.605, -415]
  MoveL 6114 to (-4.15, 71.52, -271.09) mm, rotated rx -9.61 ry -16.54 rz -54.03 deg; joints [-15.95, -56.853, 112.254, 189.089, 39.522, -110.549, -415]
  MoveL 6115 to (-2.23, 71.86, -273.73) mm, rotated rx -9.61 ry -16.54 rz -54.03 deg; joints [-16.068, -56.822, 112.335, 188.892, 39.622, -110.419, -415]
  MoveL 6116 to (-0.69, 71.49, -276.37) mm, rotated rx -9.61 ry -16.54 rz -54.03 deg; joints [-16.186, -56.836, 112.419, 188.702, 39.682, -110.298, -415]
  MoveL 6117 to (-0.25, 71.06, -277.4) mm, rotated rx -9.61 ry -16.54 rz -54.03 deg; joints [-16.232, -56.859, 112.452, 188.631, 39.687, -110.256, -415]
  MoveL 6118 to (-0.05, 70.45, -278.25) mm, rotated rx -9.61 ry -16.54 rz -54.03 deg; joints [-16.27, -56.894, 112.478, 188.575, 39.675, -110.224, -415]
  MoveL 6119 to (-0.07, 69.68, -278.91) mm, rotated rx -9.61 ry -16.54 rz -54.03 deg; joints [-16.3, -56.94, 112.498, 188.535, 39.647, -110.204, -415]
  MoveL 6120 to (-0.32, 68.74, -279.38) mm, rotated rx -9.61 ry -16.54 rz -54.03 deg; joints [-16.322, -56.997, 112.512, 188.51, 39.603, -110.195, -415]
  MoveL 6121 to (-0.79, 67.63, -279.66) mm, rotated rx -9.61 ry -16.54 rz -54.03 deg; joints [-16.335, -57.066, 112.52, 188.501, 39.541, -110.197, -415]
  MoveL 6122 to (-1.5, 66.36, -279.76) mm, rotated rx -9.61 ry -16.54 rz -54.03 deg; joints [-16.34, -57.146, 112.522, 188.507, 39.463, -110.211, -415]
  MoveL 6123 to (-1.77, 65.91, -279.76) mm, rotated rx -9.61 ry -16.54 rz -54.03 deg; joints [-16.34, -57.174, 112.522, 188.512, 39.435, -110.218, -415]
  MoveL 6124 to (-2.02, 65.51, -279.74) mm, rotated rx -9.61 ry -16.54 rz -54.03 deg; joints [-16.34, -57.199, 112.521, 188.518, 39.409, -110.224, -415]
  MoveL 6125 to (-2.25, 65.18, -279.69) mm, rotated rx -9.61 ry -16.54 rz -54.03 deg; joints [-16.338, -57.22, 112.519, 188.525, 39.387, -110.232, -415]
  MoveL 6126 to (-2.47, 64.86, -279.63) mm, rotated rx -9.61 ry -16.54 rz -54.03 deg; joints [-16.335, -57.241, 112.517, 188.533, 39.365, -110.239, -415]
  MoveL 6127 to (-2.71, 64.5, -279.59) mm, rotated rx -9.61 ry -16.54 rz -54.03 deg; joints [-16.334, -57.263, 112.515, 188.539, 39.341, -110.246, -415]
  MoveL 6128 to (-2.98, 64.09, -279.57) mm, rotated rx -9.61 ry -16.54 rz -54.03 deg; joints [-16.333, -57.289, 112.514, 188.546, 39.314, -110.253, -415]
  MoveL 6129 to (-3.25, 63.64, -279.57) mm, rotated rx -9.61 ry -16.54 rz -54.03 deg; joints [-16.333, -57.318, 112.513, 188.551, 39.286, -110.26, -415]
  MoveL 6130 to (-3.49, 63.24, -279.54) mm, rotated rx -9.61 ry -16.54 rz -54.03 deg; joints [-16.332, -57.343, 112.512, 188.556, 39.26, -110.266, -415]
  MoveL 6131 to (-3.72, 62.91, -279.49) mm, rotated rx -9.61 ry -16.54 rz -54.03 deg; joints [-16.33, -57.364, 112.511, 188.564, 39.238, -110.274, -415]
  MoveL 6132 to (-3.93, 62.58, -279.43) mm, rotated rx -9.61 ry -16.54 rz -54.03 deg; joints [-16.328, -57.385, 112.51, 188.571, 39.217, -110.281, -415]
  MoveL 6133 to (-4.17, 62.22, -279.39) mm, rotated rx -9.61 ry -16.54 rz -54.03 deg; joints [-16.326, -57.408, 112.509, 188.578, 39.193, -110.288, -415]
  MoveL 6134 to (-4.43, 61.8, -279.36) mm, rotated rx -9.61 ry -16.54 rz -54.03 deg; joints [-16.325, -57.434, 112.508, 188.585, 39.167, -110.295, -415]
  MoveL 6135 to (-4.7, 61.35, -279.36) mm, rotated rx -9.61 ry -16.54 rz -54.03 deg; joints [-16.326, -57.462, 112.508, 188.59, 39.138, -110.302, -415]
  MoveL 6136 to (-5.27, 60.55, -279.34) mm, rotated rx -9.61 ry -16.54 rz -54.03 deg; joints [-16.325, -57.512, 112.5, 188.602, 39.081, -110.316, -415]
  MoveC 6137 to (-6.09, 59.44, -279.34) mm, rotated rx -9.61 ry -16.54 rz -54.03 deg; joints [-16.324, -57.58, 112.486, 188.617, 39.001, -110.336, -415] to (-6.78, 58.24, -279.34) mm, rotated rx -9.61 ry -16.54 rz -54.03 deg; joints [-16.325, -57.655, 112.486, 188.63, 38.927, -110.353, -415]
  MoveL 6138 to (-6.78, 58.24, -279.33) mm, rotated rx -9.61 ry -16.54 rz -54.03 deg; joints [-16.325, -57.655, 112.486, 188.631, 38.927, -110.354, -415]
  MoveL 6139 to (-7.15, 57.7, -279.32) mm, rotated rx -9.61 ry -16.54 rz -54.03 deg; joints [-16.324, -57.688, 112.482, 188.639, 38.889, -110.363, -415]
  MoveL 6140 to (-7.52, 57.26, -279.29) mm, rotated rx -9.61 ry -16.54 rz -54.03 deg; joints [-16.322, -57.715, 112.473, 188.648, 38.854, -110.373, -415]
  MoveL 6141 to (-7.77, 57.08, -279.19) mm, rotated rx -9.61 ry -16.54 rz -54.03 deg; joints [-16.318, -57.726, 112.465, 188.659, 38.835, -110.382, -415]
  MoveL 6142 to (-7.76, 57.15, -278.99) mm, rotated rx -9.61 ry -16.54 rz -54.03 deg; joints [-16.309, -57.723, 112.466, 188.67, 38.84, -110.389, -415]
  MoveL 6143 to (-7.48, 57.46, -278.69) mm, rotated rx -9.61 ry -16.54 rz -54.03 deg; joints [-16.297, -57.707, 112.479, 188.683, 38.869, -110.393, -415]
  MoveL 6144 to (-7.58, 57.84, -278.06) mm, rotated rx -9.61 ry -16.54 rz -54.03 deg; joints [-16.27, -57.687, 112.466, 188.724, 38.879, -110.416, -415]
  MoveL 6145 to (-9.38, 56.87, -278.06) mm, rotated rx -9.61 ry -16.54 rz -54.03 deg; joints [-16.262, -57.736, 112.374, 188.763, 38.74, -110.458, -415]
  MoveL 6146 to (-11.31, 55.94, -278) mm, rotated rx -9.61 ry -16.54 rz -54.03 deg; joints [-16.251, -57.782, 112.271, 188.808, 38.594, -110.504, -415]
  MoveL 6147 to (-13.37, 54.98, -277.88) mm, rotated rx -9.61 ry -16.54 rz -54.03 deg; joints [-16.236, -57.828, 112.159, 188.861, 38.44, -110.557, -415]
  MoveL 6148 to (-15.4, 54.04, -277.78) mm, rotated rx -9.61 ry -16.54 rz -54.03 deg; joints [-16.222, -57.873, 112.049, 188.913, 38.288, -110.608, -415]
  MoveL 6149 to (-17.35, 53.14, -277.6) mm, rotated rx -9.61 ry -16.54 rz -54.03 deg; joints [-16.206, -57.916, 111.944, 188.967, 38.142, -110.66, -415]
  MoveL 6150 to (-19.12, 52.33, -277.46) mm, rotated rx -9.61 ry -16.54 rz -54.03 deg; joints [-16.192, -57.955, 111.848, 189.016, 38.011, -110.708, -415]
  MoveL 6151 to (-20.99, 51.46, -277.4) mm, rotated rx -9.61 ry -16.54 rz -54.03 deg; joints [-16.181, -57.995, 111.745, 189.062, 37.87, -110.755, -415]
  MoveL 6152 to (-22.95, 50.54, -277.33) mm, rotated rx -9.61 ry -16.54 rz -54.03 deg; joints [-16.169, -58.037, 111.637, 189.111, 37.724, -110.805, -415]
  MoveL 6153 to (-25.08, 49.55, -277.18) mm, rotated rx -9.61 ry -16.54 rz -54.03 deg; joints [-16.153, -58.083, 111.52, 189.169, 37.564, -110.863, -415]
  MoveL 6154 to (-26.78, 48.75, -277.07) mm, rotated rx -9.61 ry -16.54 rz -54.03 deg; joints [-16.141, -58.12, 111.427, 189.216, 37.437, -110.909, -415]
  MoveL 6155 to (-28.94, 47.74, -276.85) mm, rotated rx -9.61 ry -16.54 rz -54.03 deg; joints [-16.122, -58.166, 111.309, 189.28, 37.277, -110.97, -415]
  MoveL 6156 to (-30.64, 46.94, -276.74) mm, rotated rx -9.61 ry -16.54 rz -54.03 deg; joints [-16.11, -58.203, 111.216, 189.327, 37.15, -111.017, -415]
  MoveL 6157 to (-32.57, 46.02, -276.57) mm, rotated rx -9.61 ry -16.54 rz -54.03 deg; joints [-16.094, -58.244, 111.11, 189.383, 37.007, -111.072, -415]
  MoveL 6158 to (-34.73, 45, -276.52) mm, rotated rx -9.61 ry -16.54 rz -54.03 deg; joints [-16.082, -58.288, 110.989, 189.438, 36.844, -111.129, -415]
  MoveL 6159 to (-36.43, 44.2, -276.41) mm, rotated rx -9.61 ry -16.54 rz -54.03 deg; joints [-16.07, -58.324, 110.895, 189.486, 36.718, -111.177, -415]
  MoveL 6160 to (-38.35, 43.28, -276.25) mm, rotated rx -9.61 ry -16.54 rz -54.03 deg; joints [-16.055, -58.364, 110.788, 189.543, 36.574, -111.233, -415]
  MoveL 6161 to (-40.51, 42.25, -276.2) mm, rotated rx -9.61 ry -16.54 rz -54.03 deg; joints [-16.043, -58.408, 110.666, 189.599, 36.412, -111.291, -415]
  MoveL 6162 to (-42.21, 41.44, -276.09) mm, rotated rx -9.61 ry -16.54 rz -54.03 deg; joints [-16.031, -58.443, 110.572, 189.648, 36.286, -111.34, -415]
  MoveL 6163 to (-44.21, 40.48, -275.98) mm, rotated rx -9.61 ry -16.54 rz -54.03 deg; joints [-16.018, -58.483, 110.459, 189.705, 36.136, -111.397, -415]
  MoveL 6164 to (-46.22, 39.52, -275.92) mm, rotated rx -9.61 ry -16.54 rz -54.03 deg; joints [-16.006, -58.523, 110.345, 189.76, 35.986, -111.453, -415]
  MoveL 6165 to (-47.9, 38.68, -275.74) mm, rotated rx -9.61 ry -16.54 rz -54.03 deg; joints [-15.991, -58.56, 110.253, 189.814, 35.86, -111.506, -415]
  MoveL 6166 to (-49.44, 37.89, -275.48) mm, rotated rx -9.61 ry -16.54 rz -54.03 deg; joints [-15.975, -58.596, 110.171, 189.869, 35.746, -111.558, -415]
  MoveL 6167 to (-50.87, 37.11, -275.13) mm, rotated rx -9.61 ry -16.54 rz -54.03 deg; joints [-15.955, -58.632, 110.098, 189.928, 35.64, -111.611, -415]
  MoveL 6168 to (-49.38, 37.35, -274.44) mm, rotated rx -9.61 ry -16.54 rz -54.03 deg; joints [-15.936, -58.642, 110.215, 189.932, 35.748, -111.599, -415]
  MoveL 6169 to (-49.6, 37.29, -274.44) mm, rotated rx -9.61 ry -16.54 rz -54.03 deg; joints [-15.935, -58.644, 110.201, 189.938, 35.733, -111.605, -415]
  MoveL 6170 to (-49.9, 37.25, -274.42) mm, rotated rx -9.61 ry -16.54 rz -54.03 deg; joints [-15.932, -58.642, 110.179, 189.947, 35.713, -111.613, -415]
  MoveL 6171 to (-50.35, 37.27, -274.39) mm, rotated rx -9.61 ry -16.54 rz -54.03 deg; joints [-15.928, -58.636, 110.144, 189.961, 35.685, -111.626, -415]
  MoveL 6172 to (-50.89, 37.31, -274.35) mm, rotated rx -9.61 ry -16.54 rz -54.03 deg; joints [-15.923, -58.627, 110.102, 189.977, 35.653, -111.642, -415]
  MoveL 6173 to (-51.5, 37.37, -274.31) mm, rotated rx -9.61 ry -16.54 rz -54.03 deg; joints [-15.917, -58.615, 110.053, 189.996, 35.617, -111.659, -415]
  MoveL 6174 to (-54.09, 37.76, -274.31) mm, rotated rx -9.61 ry -16.54 rz -54.03 deg; joints [-15.898, -58.555, 109.837, 190.065, 35.465, -111.726, -415]
  MoveL 6175 to (-54.7, 37.84, -274.28) mm, rotated rx -9.61 ry -16.54 rz -54.03 deg; joints [-15.892, -58.543, 109.788, 190.084, 35.43, -111.743, -415]
  MoveL 6176 to (-55.38, 37.91, -274.22) mm, rotated rx -9.61 ry -16.54 rz -54.03 deg; joints [-15.885, -58.529, 109.733, 190.105, 35.39, -111.763, -415]
  MoveL 6177 to (-56, 37.99, -274.19) mm, rotated rx -9.61 ry -16.54 rz -54.03 deg; joints [-15.88, -58.516, 109.682, 190.124, 35.353, -111.781, -415]
  MoveL 6178 to (-56.52, 38.06, -274.19) mm, rotated rx -9.61 ry -16.54 rz -54.03 deg; joints [-15.876, -58.504, 109.639, 190.138, 35.323, -111.794, -415]
  MoveL 6179 to (-57, 38.14, -274.18) mm, rotated rx -9.61 ry -16.54 rz -54.03 deg; joints [-15.872, -58.493, 109.598, 190.152, 35.294, -111.807, -415]
  MoveL 6180 to (-57.52, 38.22, -274.18) mm, rotated rx -9.61 ry -16.54 rz -54.03 deg; joints [-15.868, -58.481, 109.555, 190.166, 35.264, -111.821, -415]
  MoveL 6181 to (-58.03, 38.29, -274.18) mm, rotated rx -9.61 ry -16.54 rz -54.03 deg; joints [-15.864, -58.469, 109.512, 190.18, 35.234, -111.834, -415]
  MoveL 6182 to (-58.51, 38.35, -274.15) mm, rotated rx -9.61 ry -16.54 rz -54.03 deg; joints [-15.86, -58.459, 109.473, 190.194, 35.206, -111.848, -415]
  MoveL 6183 to (-58.97, 38.4, -274.1) mm, rotated rx -9.61 ry -16.54 rz -54.03 deg; joints [-15.855, -58.45, 109.436, 190.21, 35.179, -111.862, -415]
  MoveL 6184 to (-59.46, 38.47, -274.09) mm, rotated rx -9.61 ry -16.54 rz -54.03 deg; joints [-15.851, -58.439, 109.395, 190.224, 35.15, -111.876, -415]
  MoveL 6185 to (-59.99, 38.55, -274.08) mm, rotated rx -9.61 ry -16.54 rz -54.03 deg; joints [-15.847, -58.427, 109.351, 190.239, 35.119, -111.89, -415]
  MoveL 6186 to (-61.03, 38.7, -274.08) mm, rotated rx -9.61 ry -16.54 rz -54.03 deg; joints [-15.839, -58.403, 109.264, 190.267, 35.059, -111.917, -415]
  Set speed (1000.0 mm/s)
  MoveL 6187 to (-80.62, 47.84, -274.08) mm, rotated rx -9.61 ry -16.54 rz -54.03 deg; joints [-15.673, -57.523, 107.356, 190.82, 34.066, -112.433, -415]
  Print: /'Flow1'
  Set speed (1000.0 mm/s)
  MoveL 6188 to (-40.38, -104.96, -81.82) mm, rotated rx 105.8 ry 33.04 rz 34.05 deg; joints [-3.332, -28.971, 98.058, 147.608, 81.185, 20.391, -475]
  Set speed (1000.0 mm/s)
  MoveL 6189 to (-3.62, -79.22, -81.82) mm, rotated rx 105.8 ry 33.04 rz 34.05 deg; joints [-3.3, -29.88, 101.913, 147.848, 83.67, 18.796, -475]
  Set speed (100.0 mm/s)
  MoveL 6190 to (55.98, -37.48, -81.82) mm, rotated rx 105.8 ry 33.04 rz 34.05 deg; joints [-3.244, -31.04, 107.839, 148.094, 87.703, 16.249, -475]
  MoveL 6191 to (56.51, -37.51, -81.82) mm, rotated rx 105.8 ry 33.04 rz 34.05 deg; joints [-3.243, -31.067, 107.885, 148.095, 87.72, 16.238, -475]
  MoveL 6192 to (57.15, -37.49, -81.72) mm, rotated rx 105.8 ry 33.04 rz 34.05 deg; joints [-3.239, -31.098, 107.943, 148.1, 87.743, 16.223, -475]
  MoveL 6193 to (57.74, -37.49, -81.67) mm, rotated rx 105.8 ry 33.04 rz 34.05 deg; joints [-3.236, -31.127, 107.996, 148.104, 87.763, 16.21, -475]
  MoveL 6194 to (58.31, -37.51, -81.64) mm, rotated rx 105.8 ry 33.04 rz 34.05 deg; joints [-3.234, -31.155, 108.047, 148.106, 87.781, 16.198, -475]
  MoveL 6195 to (61.97, -37.71, -81.64) mm, rotated rx 105.8 ry 33.04 rz 34.05 deg; joints [-3.231, -31.344, 108.373, 148.112, 87.897, 16.125, -475]
  MoveL 6196 to (63.41, -37.85, -81.73) mm, rotated rx 105.8 ry 33.04 rz 34.05 deg; joints [-3.233, -31.422, 108.501, 148.111, 87.941, 16.098, -475]
  MoveL 6197 to (64.57, -38.09, -82) mm, rotated rx 105.8 ry 33.04 rz 34.05 deg; joints [-3.242, -31.491, 108.603, 148.102, 87.97, 16.082, -475]
  MoveL 6198 to (65.45, -38.45, -82.44) mm, rotated rx 105.8 ry 33.04 rz 34.05 deg; joints [-3.26, -31.551, 108.68, 148.085, 87.986, 16.077, -475]
  MoveL 6199 to (65.79, -38.66, -82.73) mm, rotated rx 105.8 ry 33.04 rz 34.05 deg; joints [-3.271, -31.578, 108.708, 148.074, 87.988, 16.079, -475]
  MoveL 6200 to (66.05, -38.9, -83.06) mm, rotated rx 105.8 ry 33.04 rz 34.05 deg; joints [-3.285, -31.603, 108.73, 148.061, 87.987, 16.083, -475]
  MoveL 6201 to (66.37, -39.46, -83.86) mm, rotated rx 105.8 ry 33.04 rz 34.05 deg; joints [-3.317, -31.646, 108.755, 148.029, 87.975, 16.098, -475]
  MoveL 6202 to (66.4, -40.13, -84.84) mm, rotated rx 105.8 ry 33.04 rz 34.05 deg; joints [-3.357, -31.68, 108.753, 147.989, 87.95, 16.125, -475]
  MoveL 6203 to (65.62, -41.79, -87.32) mm, rotated rx 105.8 ry 33.04 rz 34.05 deg; joints [-3.459, -31.723, 108.673, 147.886, 87.857, 16.21, -475]
  MoveL 6204 to (64.05, -43.35, -89.81) mm, rotated rx 105.8 ry 33.04 rz 34.05 deg; joints [-3.562, -31.723, 108.522, 147.782, 87.743, 16.31, -475]
  MoveL 6205 to (62.03, -44.32, -91.58) mm, rotated rx 105.8 ry 33.04 rz 34.05 deg; joints [-3.636, -31.671, 108.335, 147.707, 87.638, 16.396, -475]
  MoveL 6206 to (60.86, -44.58, -92.2) mm, rotated rx 105.8 ry 33.04 rz 34.05 deg; joints [-3.662, -31.626, 108.229, 147.68, 87.589, 16.434, -475]
  MoveL 6207 to (59.57, -44.68, -92.65) mm, rotated rx 105.8 ry 33.04 rz 34.05 deg; joints [-3.681, -31.568, 108.113, 147.66, 87.543, 16.469, -475]
  MoveL 6208 to (56.67, -44.45, -93) mm, rotated rx 105.8 ry 33.04 rz 34.05 deg; joints [-3.698, -31.413, 107.855, 147.641, 87.457, 16.528, -475]
  MoveL 6209 to (53.56, -43.92, -93.01) mm, rotated rx 105.8 ry 33.04 rz 34.05 deg; joints [-3.7, -31.235, 107.581, 147.636, 87.377, 16.58, -475]
  MoveL 6210 to (53.08, -43.85, -93.03) mm, rotated rx 105.8 ry 33.04 rz 34.05 deg; joints [-3.701, -31.208, 107.538, 147.635, 87.363, 16.588, -475]
  MoveL 6211 to (52.62, -43.8, -93.07) mm, rotated rx 105.8 ry 33.04 rz 34.05 deg; joints [-3.703, -31.183, 107.498, 147.632, 87.351, 16.597, -475]
  MoveL 6212 to (52.21, -43.77, -93.13) mm, rotated rx 105.8 ry 33.04 rz 34.05 deg; joints [-3.706, -31.161, 107.461, 147.629, 87.338, 16.606, -475]
  MoveL 6213 to (51.76, -43.73, -93.18) mm, rotated rx 105.8 ry 33.04 rz 34.05 deg; joints [-3.708, -31.137, 107.421, 147.627, 87.325, 16.614, -475]
  MoveL 6214 to (51.22, -43.65, -93.2) mm, rotated rx 105.8 ry 33.04 rz 34.05 deg; joints [-3.71, -31.107, 107.373, 147.625, 87.311, 16.624, -475]
  MoveL 6215 to (50.58, -43.56, -93.24) mm, rotated rx 105.8 ry 33.04 rz 34.05 deg; joints [-3.712, -31.071, 107.316, 147.622, 87.293, 16.636, -475]
  MoveL 6216 to (50.02, -43.5, -93.3) mm, rotated rx 105.8 ry 33.04 rz 34.05 deg; joints [-3.715, -31.041, 107.267, 147.619, 87.277, 16.647, -475]
  MoveL 6217 to (49.58, -43.47, -93.37) mm, rotated rx 105.8 ry 33.04 rz 34.05 deg; joints [-3.718, -31.017, 107.227, 147.615, 87.264, 16.656, -475]
  MoveL 6218 to (49.14, -43.43, -93.42) mm, rotated rx 105.8 ry 33.04 rz 34.05 deg; joints [-3.72, -30.994, 107.188, 147.613, 87.251, 16.665, -475]
  MoveL 6219 to (48.67, -43.36, -93.45) mm, rotated rx 105.8 ry 33.04 rz 34.05 deg; joints [-3.721, -30.967, 107.146, 147.611, 87.238, 16.673, -475]
  MoveL 6220 to (48.15, -43.27, -93.45) mm, rotated rx 105.8 ry 33.04 rz 34.05 deg; joints [-3.722, -30.937, 107.1, 147.61, 87.225, 16.682, -475]
  MoveL 6221 to (47.62, -43.18, -93.45) mm, rotated rx 105.8 ry 33.04 rz 34.05 deg; joints [-3.722, -30.907, 107.053, 147.61, 87.211, 16.691, -475]
  MoveL 6222 to (47.05, -43.1, -93.46) mm, rotated rx 105.8 ry 33.04 rz 34.05 deg; joints [-3.723, -30.875, 107.003, 147.608, 87.195, 16.701, -475]
  MoveL 6223 to (46.4, -43.02, -93.49) mm, rotated rx 105.8 ry 33.04 rz 34.05 deg; joints [-3.725, -30.839, 106.944, 147.606, 87.176, 16.714, -475]
  MoveL 6224 to (45.81, -42.98, -93.56) mm, rotated rx 105.8 ry 33.04 rz 34.05 deg; joints [-3.728, -30.808, 106.891, 147.602, 87.158, 16.726, -475]
  MoveL 6225 to (45.35, -42.98, -93.66) mm, rotated rx 105.8 ry 33.04 rz 34.05 deg; joints [-3.732, -30.785, 106.85, 147.597, 87.143, 16.737, -475]
  MoveL 6226 to (45.35, -42.97, -93.9) mm, rotated rx 105.8 ry 33.04 rz 34.05 deg; joints [-3.742, -30.785, 106.851, 147.588, 87.145, 16.738, -475]
  MoveL 6227 to (45.75, -42.91, -94.25) mm, rotated rx 105.8 ry 33.04 rz 34.05 deg; joints [-3.756, -30.802, 106.887, 147.575, 87.163, 16.731, -475]
  MoveL 6228 to (46.36, -43.5, -95.22) mm, rotated rx 105.8 ry 33.04 rz 34.05 deg; joints [-3.795, -30.861, 106.938, 147.537, 87.162, 16.743, -475]
  MoveL 6229 to (44.41, -44.37, -95.22) mm, rotated rx 105.8 ry 33.04 rz 34.05 deg; joints [-3.796, -30.804, 106.753, 147.532, 87.054, 16.812, -475]
  MoveL 6230 to (42.33, -45.34, -95.35) mm, rotated rx 105.8 ry 33.04 rz 34.05 deg; joints [-3.802, -30.746, 106.556, 147.522, 86.937, 16.888, -475]
  MoveL 6231 to (40.35, -46.24, -95.4) mm, rotated rx 105.8 ry 33.04 rz 34.05 deg; joints [-3.806, -30.688, 106.367, 147.515, 86.827, 16.959, -475]
  MoveL 6232 to (38.42, -47.13, -95.53) mm, rotated rx 105.8 ry 33.04 rz 34.05 deg; joints [-3.812, -30.633, 106.183, 147.505, 86.719, 17.03, -475]
  MoveL 6233 to (36.47, -48.02, -95.69) mm, rotated rx 105.8 ry 33.04 rz 34.05 deg; joints [-3.819, -30.577, 105.997, 147.494, 86.611, 17.101, -475]
  MoveL 6234 to (34.54, -48.9, -95.81) mm, rotated rx 105.8 ry 33.04 rz 34.05 deg; joints [-3.825, -30.52, 105.812, 147.483, 86.503, 17.172, -475]
  MoveL 6235 to (32.59, -49.8, -96.02) mm, rotated rx 105.8 ry 33.04 rz 34.05 deg; joints [-3.834, -30.463, 105.625, 147.47, 86.395, 17.243, -475]
  MoveL 6236 to (30.66, -50.68, -96.14) mm, rotated rx 105.8 ry 33.04 rz 34.05 deg; joints [-3.84, -30.406, 105.44, 147.46, 86.288, 17.314, -475]
  MoveL 6237 to (28.7, -51.56, -96.19) mm, rotated rx 105.8 ry 33.04 rz 34.05 deg; joints [-3.843, -30.347, 105.251, 147.452, 86.179, 17.384, -475]
  MoveL 6238 to (26.73, -52.44, -96.34) mm, rotated rx 105.8 ry 33.04 rz 34.05 deg; joints [-3.85, -30.288, 105.062, 147.441, 86.071, 17.456, -475]
  MoveL 6239 to (24.7, -53.36, -96.52) mm, rotated rx 105.8 ry 33.04 rz 34.05 deg; joints [-3.858, -30.227, 104.866, 147.428, 85.958, 17.53, -475]
  MoveL 6240 to (22.67, -54.26, -96.7) mm, rotated rx 105.8 ry 33.04 rz 34.05 deg; joints [-3.867, -30.164, 104.67, 147.415, 85.847, 17.605, -475]
  MoveL 6241 to (20.95, -55.02, -96.94) mm, rotated rx 105.8 ry 33.04 rz 34.05 deg; joints [-3.877, -30.112, 104.505, 147.4, 85.753, 17.668, -475]
  MoveL 6242 to (18.52, -56.11, -97.05) mm, rotated rx 105.8 ry 33.04 rz 34.05 deg; joints [-3.882, -30.036, 104.268, 147.388, 85.618, 17.756, -475]
  Set speed (1000.0 mm/s)
  MoveL 6243 to (-18.59, -82.09, -97.05) mm, rotated rx 105.8 ry 33.04 rz 34.05 deg; joints [-3.898, -29.23, 100.489, 147.214, 83.119, 19.374, -475]
  Set speed (1000.0 mm/s)
  MoveL 6244 to (-21.88, -77.39, -108.93) mm, rotated rx 105.8 ry 33.04 rz 34.05 deg; joints [-4.357, -28.869, 100.245, 146.773, 83.297, 19.434, -475]
  Set speed (100.0 mm/s)
  MoveL 6245 to (1.62, -60.94, -108.93) mm, rotated rx 105.8 ry 33.04 rz 34.05 deg; joints [-4.356, -29.394, 102.657, 146.881, 84.876, 18.395, -475]
  MoveL 6246 to (3.27, -60.46, -108.68) mm, rotated rx 105.8 ry 33.04 rz 34.05 deg; joints [-4.346, -29.458, 102.816, 146.895, 84.954, 18.341, -475]
  MoveL 6247 to (5.2, -59.86, -108.62) mm, rotated rx 105.8 ry 33.04 rz 34.05 deg; joints [-4.343, -29.531, 103.003, 146.904, 85.049, 18.278, -475]
  MoveL 6248 to (7.16, -59.26, -108.47) mm, rotated rx 105.8 ry 33.04 rz 34.05 deg; joints [-4.337, -29.605, 103.192, 146.915, 85.145, 18.213, -475]
  MoveL 6249 to (9.52, -58.55, -108.34) mm, rotated rx 105.8 ry 33.04 rz 34.05 deg; joints [-4.331, -29.695, 103.419, 146.927, 85.259, 18.137, -475]
  MoveL 6250 to (11.56, -57.92, -108.34) mm, rotated rx 105.8 ry 33.04 rz 34.05 deg; joints [-4.331, -29.771, 103.615, 146.932, 85.359, 18.071, -475]
  MoveL 6251 to (13.81, -57.21, -108.18) mm, rotated rx 105.8 ry 33.04 rz 34.05 deg; joints [-4.324, -29.855, 103.832, 146.945, 85.469, 17.997, -475]
  MoveL 6252 to (15.71, -56.63, -108) mm, rotated rx 105.8 ry 33.04 rz 34.05 deg; joints [-4.316, -29.926, 104.014, 146.957, 85.561, 17.934, -475]
  MoveL 6253 to (17.67, -56.03, -107.9) mm, rotated rx 105.8 ry 33.04 rz 34.05 deg; joints [-4.312, -29.999, 104.202, 146.966, 85.657, 17.871, -475]
  MoveL 6254 to (19.71, -55.39, -107.69) mm, rotated rx 105.8 ry 33.04 rz 34.05 deg; joints [-4.303, -30.074, 104.396, 146.98, 85.756, 17.803, -475]
  MoveL 6255 to (21.72, -54.76, -107.53) mm, rotated rx 105.8 ry 33.04 rz 34.05 deg; joints [-4.296, -30.148, 104.588, 146.991, 85.854, 17.737, -475]
  MoveL 6256 to (23.74, -54.12, -107.42) mm, rotated rx 105.8 ry 33.04 rz 34.05 deg; joints [-4.292, -30.221, 104.781, 147, 85.953, 17.671, -475]
  MoveL 6257 to (25.78, -53.47, -107.25) mm, rotated rx 105.8 ry 33.04 rz 34.05 deg; joints [-4.285, -30.295, 104.975, 147.012, 86.053, 17.604, -475]
  MoveL 6258 to (27.8, -52.82, -107.11) mm, rotated rx 105.8 ry 33.04 rz 34.05 deg; joints [-4.278, -30.368, 105.167, 147.022, 86.152, 17.537, -475]
  MoveL 6259 to (29.88, -52.17, -107.04) mm, rotated rx 105.8 ry 33.04 rz 34.05 deg; joints [-4.275, -30.444, 105.364, 147.03, 86.254, 17.47, -475]
  MoveL 6260 to (31.91, -51.5, -106.83) mm, rotated rx 105.8 ry 33.04 rz 34.05 deg; joints [-4.267, -30.515, 105.556, 147.042, 86.354, 17.403, -475]
  MoveL 6261 to (33.92, -50.85, -106.71) mm, rotated rx 105.8 ry 33.04 rz 34.05 deg; joints [-4.261, -30.587, 105.747, 147.052, 86.453, 17.337, -475]
  MoveL 6262 to (35.98, -50.18, -106.59) mm, rotated rx 105.8 ry 33.04 rz 34.05 deg; joints [-4.256, -30.66, 105.942, 147.061, 86.554, 17.269, -475]
  MoveL 6263 to (37.62, -49.51, -106.38) mm, rotated rx 105.8 ry 33.04 rz 34.05 deg; joints [-4.247, -30.712, 106.098, 147.073, 86.64, 17.211, -475]
  MoveL 6264 to (38.93, -48.83, -106.03) mm, rotated rx 105.8 ry 33.04 rz 34.05 deg; joints [-4.233, -30.746, 106.223, 147.09, 86.715, 17.158, -475]
  MoveL 6265 to (39.9, -48.11, -105.5) mm, rotated rx 105.8 ry 33.04 rz 34.05 deg; joints [-4.211, -30.761, 106.318, 147.113, 86.779, 17.11, -475]
  MoveL 6266 to (38.36, -48.11, -104.64) mm, rotated rx 105.8 ry 33.04 rz 34.05 deg; joints [-4.177, -30.683, 106.178, 147.145, 86.722, 17.137, -475]
  MoveL 6267 to (39.16, -48.04, -104.64) mm, rotated rx 105.8 ry 33.04 rz 34.05 deg; joints [-4.177, -30.72, 106.251, 147.146, 86.753, 17.117, -475]
  MoveL 6268 to (39.86, -48.04, -104.64) mm, rotated rx 105.8 ry 33.04 rz 34.05 deg; joints [-4.177, -30.755, 106.315, 147.147, 86.777, 17.101, -475]
  MoveL 6269 to (40.49, -48.14, -104.64) mm, rotated rx 105.8 ry 33.04 rz 34.05 deg; joints [-4.176, -30.791, 106.371, 147.148, 86.794, 17.09, -475]
  MoveL 6270 to (41.14, -48.28, -104.62) mm, rotated rx 105.8 ry 33.04 rz 34.05 deg; joints [-4.175, -30.83, 106.429, 147.15, 86.809, 17.08, -475]
  MoveL 6271 to (41.89, -48.47, -104.58) mm, rotated rx 105.8 ry 33.04 rz 34.05 deg; joints [-4.174, -30.876, 106.494, 147.152, 86.826, 17.069, -475]
  MoveL 6272 to (43.89, -49.07, -104.58) mm, rotated rx 105.8 ry 33.04 rz 34.05 deg; joints [-4.173, -31.004, 106.671, 147.155, 86.866, 17.042, -475]
  MoveL 6273 to (44.32, -49.18, -104.56) mm, rotated rx 105.8 ry 33.04 rz 34.05 deg; joints [-4.172, -31.03, 106.708, 147.156, 86.875, 17.036, -475]
  MoveL 6274 to (45.33, -49.48, -104.56) mm, rotated rx 105.8 ry 33.04 rz 34.05 deg; joints [-4.171, -31.094, 106.796, 147.157, 86.895, 17.023, -475]
  MoveL 6275 to (45.81, -49.62, -104.56) mm, rotated rx 105.8 ry 33.04 rz 34.05 deg; joints [-4.171, -31.125, 106.839, 147.158, 86.905, 17.016, -475]
  MoveL 6276 to (46.29, -49.75, -104.54) mm, rotated rx 105.8 ry 33.04 rz 34.05 deg; joints [-4.17, -31.154, 106.88, 147.159, 86.915, 17.01, -475]
  MoveL 6277 to (46.75, -49.87, -104.51) mm, rotated rx 105.8 ry 33.04 rz 34.05 deg; joints [-4.168, -31.183, 106.921, 147.161, 86.925, 17.003, -475]
  MoveL 6278 to (47.18, -49.95, -104.45) mm, rotated rx 105.8 ry 33.04 rz 34.05 deg; joints [-4.166, -31.208, 106.959, 147.164, 86.936, 16.995, -475]
  MoveL 6279 to (47.64, -50.06, -104.41) mm, rotated rx 105.8 ry 33.04 rz 34.05 deg; joints [-4.164, -31.236, 106.999, 147.166, 86.946, 16.988, -475]
  MoveL 6280 to (48.11, -50.19, -104.39) mm, rotated rx 105.8 ry 33.04 rz 34.05 deg; joints [-4.163, -31.266, 107.041, 147.167, 86.956, 16.982, -475]
  MoveL 6281 to (48.6, -50.33, -104.39) mm, rotated rx 105.8 ry 33.04 rz 34.05 deg; joints [-4.162, -31.297, 107.084, 147.168, 86.966, 16.975, -475]
  MoveL 6282 to (49.08, -50.46, -104.37) mm, rotated rx 105.8 ry 33.04 rz 34.05 deg; joints [-4.161, -31.326, 107.125, 147.17, 86.976, 16.968, -475]
  MoveL 6283 to (49.55, -50.57, -104.33) mm, rotated rx 105.8 ry 33.04 rz 34.05 deg; joints [-4.16, -31.355, 107.166, 147.171, 86.986, 16.961, -475]
  MoveL 6284 to (49.97, -50.65, -104.28) mm, rotated rx 105.8 ry 33.04 rz 34.05 deg; joints [-4.157, -31.379, 107.204, 147.174, 86.996, 16.954, -475]
  MoveL 6285 to (50.42, -50.74, -104.22) mm, rotated rx 105.8 ry 33.04 rz 34.05 deg; joints [-4.155, -31.406, 107.243, 147.177, 87.007, 16.946, -475]
  MoveL 6286 to (51.82, -51.08, -104.14) mm, rotated rx 105.8 ry 33.04 rz 34.05 deg; joints [-4.151, -31.491, 107.366, 147.182, 87.038, 16.925, -475]
  MoveL 6287 to (52.92, -51.5, -104.27) mm, rotated rx 105.8 ry 33.04 rz 34.05 deg; joints [-4.155, -31.566, 107.46, 147.178, 87.055, 16.915, -475]
  MoveL 6288 to (53.72, -52, -104.6) mm, rotated rx 105.8 ry 33.04 rz 34.05 deg; joints [-4.169, -31.629, 107.528, 147.165, 87.06, 16.916, -475]
  MoveL 6289 to (54, -52.28, -104.85) mm, rotated rx 105.8 ry 33.04 rz 34.05 deg; joints [-4.178, -31.656, 107.551, 147.155, 87.058, 16.92, -475]
  MoveL 6290 to (54.22, -52.58, -105.15) mm, rotated rx 105.8 ry 33.04 rz 34.05 deg; joints [-4.19, -31.681, 107.567, 147.143, 87.053, 16.927, -475]
  MoveL 6291 to (54.42, -53.24, -105.91) mm, rotated rx 105.8 ry 33.04 rz 34.05 deg; joints [-4.221, -31.722, 107.579, 147.113, 87.032, 16.949, -475]
  MoveL 6292 to (54.33, -53.97, -106.88) mm, rotated rx 105.8 ry 33.04 rz 34.05 deg; joints [-4.26, -31.752, 107.564, 147.073, 87, 16.981, -475]
  MoveL 6293 to (53.25, -55.66, -109.44) mm, rotated rx 105.8 ry 33.04 rz 34.05 deg; joints [-4.363, -31.778, 107.45, 146.968, 86.896, 17.079, -475]
  MoveL 6294 to (51.41, -57.12, -112.05) mm, rotated rx 105.8 ry 33.04 rz 34.05 deg; joints [-4.469, -31.755, 107.27, 146.86, 86.779, 17.187, -475]
  MoveL 6295 to (50.38, -57.56, -113.08) mm, rotated rx 105.8 ry 33.04 rz 34.05 deg; joints [-4.511, -31.724, 107.173, 146.817, 86.729, 17.232, -475]
  MoveL 6296 to (49.27, -57.81, -113.92) mm, rotated rx 105.8 ry 33.04 rz 34.05 deg; joints [-4.544, -31.68, 107.071, 146.782, 86.685, 17.271, -475]
  MoveL 6297 to (48.09, -57.85, -114.57) mm, rotated rx 105.8 ry 33.04 rz 34.05 deg; joints [-4.571, -31.623, 106.963, 146.754, 86.646, 17.305, -475]
  MoveL 6298 to (46.82, -57.71, -115.04) mm, rotated rx 105.8 ry 33.04 rz 34.05 deg; joints [-4.59, -31.553, 106.851, 146.734, 86.613, 17.332, -475]
  MoveL 6299 to (45.48, -57.37, -115.32) mm, rotated rx 105.8 ry 33.04 rz 34.05 deg; joints [-4.602, -31.471, 106.733, 146.722, 86.586, 17.354, -475]
  MoveL 6300 to (44.07, -56.83, -115.41) mm, rotated rx 105.8 ry 33.04 rz 34.05 deg; joints [-4.606, -31.375, 106.611, 146.717, 86.564, 17.369, -475]
  MoveL 6301 to (41.17, -55.57, -115.41) mm, rotated rx 105.8 ry 33.04 rz 34.05 deg; joints [-4.607, -31.172, 106.361, 146.714, 86.525, 17.395, -475]
  MoveL 6302 to (40.66, -55.36, -115.43) mm, rotated rx 105.8 ry 33.04 rz 34.05 deg; joints [-4.607, -31.137, 106.317, 146.713, 86.518, 17.4, -475]
  MoveL 6303 to (40.08, -55.13, -115.46) mm, rotated rx 105.8 ry 33.04 rz 34.05 deg; joints [-4.609, -31.097, 106.267, 146.711, 86.509, 17.406, -475]
  MoveL 6304 to (39.36, -54.89, -115.56) mm, rotated rx 105.8 ry 33.04 rz 34.05 deg; joints [-4.613, -31.05, 106.204, 146.707, 86.497, 17.416, -475]
  MoveL 6305 to (38.78, -54.66, -115.59) mm, rotated rx 105.8 ry 33.04 rz 34.05 deg; joints [-4.615, -31.011, 106.154, 146.705, 86.488, 17.422, -475]
  MoveL 6306 to (38.28, -54.45, -115.61) mm, rotated rx 105.8 ry 33.04 rz 34.05 deg; joints [-4.615, -30.976, 106.111, 146.704, 86.481, 17.427, -475]
  MoveL 6307 to (37.81, -54.26, -115.62) mm, rotated rx 105.8 ry 33.04 rz 34.05 deg; joints [-4.616, -30.944, 106.07, 146.703, 86.474, 17.431, -475]
  MoveL 6308 to (37.39, -54.08, -115.63) mm, rotated rx 105.8 ry 33.04 rz 34.05 deg; joints [-4.616, -30.914, 106.033, 146.702, 86.468, 17.436, -475]
  MoveL 6309 to (35.5, -53.27, -115.64) mm, rotated rx 105.8 ry 33.04 rz 34.05 deg; joints [-4.617, -30.782, 105.87, 146.7, 86.442, 17.453, -475]
  MoveL 6310 to (35.02, -53.09, -115.68) mm, rotated rx 105.8 ry 33.04 rz 34.05 deg; joints [-4.619, -30.75, 105.828, 146.698, 86.434, 17.459, -475]
  MoveL 6311 to (34.57, -52.93, -115.73) mm, rotated rx 105.8 ry 33.04 rz 34.05 deg; joints [-4.621, -30.721, 105.789, 146.696, 86.426, 17.465, -475]
  MoveL 6312 to (34.13, -52.8, -115.8) mm, rotated rx 105.8 ry 33.04 rz 34.05 deg; joints [-4.624, -30.692, 105.75, 146.693, 86.418, 17.471, -475]
  MoveL 6313 to (33.66, -52.68, -115.86) mm, rotated rx 105.8 ry 33.04 rz 34.05 deg; joints [-4.627, -30.663, 105.708, 146.69, 86.408, 17.479, -475]
  MoveL 6314 to (33.12, -52.56, -115.89) mm, rotated rx 105.8 ry 33.04 rz 34.05 deg; joints [-4.628, -30.631, 105.66, 146.688, 86.395, 17.487, -475]
  MoveL 6315 to (32.45, -52.51, -115.9) mm, rotated rx 105.8 ry 33.04 rz 34.05 deg; joints [-4.628, -30.595, 105.599, 146.687, 86.374, 17.501, -475]
  MoveL 6316 to (31.68, -52.52, -115.9) mm, rotated rx 105.8 ry 33.04 rz 34.05 deg; joints [-4.629, -30.556, 105.529, 146.685, 86.347, 17.519, -475]
  MoveL 6317 to (33.4, -53.42, -117.46) mm, rotated rx 105.8 ry 33.04 rz 34.05 deg; joints [-4.69, -30.684, 105.677, 146.626, 86.373, 17.521, -475]
  MoveL 6318 to (31.08, -53.87, -117.59) mm, rotated rx 105.8 ry 33.04 rz 34.05 deg; joints [-4.695, -30.588, 105.46, 146.616, 86.273, 17.589, -475]
  MoveL 6319 to (28.88, -54.29, -117.7) mm, rotated rx 105.8 ry 33.04 rz 34.05 deg; joints [-4.7, -30.496, 105.255, 146.608, 86.179, 17.652, -475]
  MoveL 6320 to (26.77, -54.71, -117.86) mm, rotated rx 105.8 ry 33.04 rz 34.05 deg; joints [-4.706, -30.408, 105.056, 146.598, 86.088, 17.715, -475]
  MoveL 6321 to (24.67, -55.11, -117.97) mm, rotated rx 105.8 ry 33.04 rz 34.05 deg; joints [-4.71, -30.32, 104.86, 146.589, 85.998, 17.775, -475]
  MoveL 6322 to (22.57, -55.51, -118.08) mm, rotated rx 105.8 ry 33.04 rz 34.05 deg; joints [-4.715, -30.231, 104.662, 146.581, 85.907, 17.836, -475]
  MoveL 6323 to (20.48, -55.92, -118.3) mm, rotated rx 105.8 ry 33.04 rz 34.05 deg; joints [-4.723, -30.144, 104.465, 146.568, 85.817, 17.899, -475]
  MoveL 6324 to (18.38, -56.33, -118.52) mm, rotated rx 105.8 ry 33.04 rz 34.05 deg; joints [-4.732, -30.055, 104.267, 146.555, 85.727, 17.961, -475]
  MoveL 6325 to (16.28, -56.72, -118.64) mm, rotated rx 105.8 ry 33.04 rz 34.05 deg; joints [-4.736, -29.966, 104.069, 146.546, 85.637, 18.022, -475]
  MoveL 6326 to (14.18, -57.1, -118.64) mm, rotated rx 105.8 ry 33.04 rz 34.05 deg; joints [-4.736, -29.876, 103.871, 146.542, 85.547, 18.082, -475]
  MoveL 6327 to (12.08, -57.49, -118.75) mm, rotated rx 105.8 ry 33.04 rz 34.05 deg; joints [-4.741, -29.786, 103.672, 146.533, 85.457, 18.143, -475]
  MoveL 6328 to (9.96, -57.88, -118.95) mm, rotated rx 105.8 ry 33.04 rz 34.05 deg; joints [-4.749, -29.694, 103.47, 146.52, 85.366, 18.206, -475]
  MoveL 6329 to (7.97, -58.24, -119.13) mm, rotated rx 105.8 ry 33.04 rz 34.05 deg; joints [-4.756, -29.609, 103.282, 146.509, 85.281, 18.265, -475]
  MoveL 6330 to (6.15, -58.58, -119.35) mm, rotated rx 105.8 ry 33.04 rz 34.05 deg; joints [-4.764, -29.53, 103.108, 146.496, 85.204, 18.319, -475]
  MoveL 6331 to (4.22, -58.93, -119.44) mm, rotated rx 105.8 ry 33.04 rz 34.05 deg; joints [-4.767, -29.446, 102.924, 146.488, 85.12, 18.376, -475]
  MoveL 6332 to (2.16, -59.3, -119.45) mm, rotated rx 105.8 ry 33.04 rz 34.05 deg; joints [-4.768, -29.357, 102.728, 146.483, 85.031, 18.435, -475]
  MoveL 6333 to (-0.51, -59.77, -119.55) mm, rotated rx 105.8 ry 33.04 rz 34.05 deg; joints [-4.771, -29.24, 102.473, 146.472, 84.917, 18.512, -475]
  MoveL 6334 to (-2.52, -60.11, -119.76) mm, rotated rx 105.8 ry 33.04 rz 34.05 deg; joints [-4.779, -29.151, 102.281, 146.459, 84.832, 18.572, -475]
  MoveL 6335 to (-4.69, -60.48, -119.96) mm, rotated rx 105.8 ry 33.04 rz 34.05 deg; joints [-4.787, -29.055, 102.073, 146.446, 84.74, 18.636, -475]
  MoveL 6336 to (-6.69, -60.8, -120.25) mm, rotated rx 105.8 ry 33.04 rz 34.05 deg; joints [-4.798, -28.966, 101.881, 146.43, 84.657, 18.695, -475]
  MoveL 6337 to (-8.64, -61.14, -120.38) mm, rotated rx 105.8 ry 33.04 rz 34.05 deg; joints [-4.803, -28.879, 101.693, 146.42, 84.573, 18.753, -475]
  MoveL 6338 to (-10.7, -61.51, -120.39) mm, rotated rx 105.8 ry 33.04 rz 34.05 deg; joints [-4.803, -28.789, 101.495, 146.414, 84.483, 18.813, -475]
  MoveL 6339 to (-12.45, -61.78, -120.62) mm, rotated rx 105.8 ry 33.04 rz 34.05 deg; joints [-4.812, -28.709, 101.326, 146.401, 84.41, 18.864, -475]
  Set speed (1000.0 mm/s)
  MoveL 6340 to (-33.8, -76.72, -120.62) mm, rotated rx 105.8 ry 33.04 rz 34.05 deg; joints [-4.805, -28.216, 99.114, 146.302, 82.978, 19.821, -475]
  Set speed (1000.0 mm/s)
  MoveL 6341 to (-37.55, -71.37, -131.81) mm, rotated rx 105.8 ry 33.04 rz 34.05 deg; joints [-5.233, -27.799, 98.812, 145.891, 83.151, 19.873, -475]
  Set speed (100.0 mm/s)
  MoveL 6342 to (-21.02, -59.8, -131.81) mm, rotated rx 105.8 ry 33.04 rz 34.05 deg; joints [-5.244, -28.182, 100.529, 145.963, 84.258, 19.124, -475]
  MoveL 6343 to (-18.89, -59.68, -131.81) mm, rotated rx 105.8 ry 33.04 rz 34.05 deg; joints [-5.245, -28.288, 100.733, 145.968, 84.339, 19.069, -475]
  MoveL 6344 to (-16.66, -59.58, -131.71) mm, rotated rx 105.8 ry 33.04 rz 34.05 deg; joints [-5.242, -28.4, 100.946, 145.976, 84.423, 19.012, -475]
  MoveL 6345 to (-14.32, -59.52, -131.42) mm, rotated rx 105.8 ry 33.04 rz 34.05 deg; joints [-5.231, -28.519, 101.169, 145.992, 84.508, 18.95, -475]
  MoveL 6346 to (-12.07, -59.46, -131.07) mm, rotated rx 105.8 ry 33.04 rz 34.05 deg; joints [-5.218, -28.633, 101.383, 146.01, 84.588, 18.891, -475]
  MoveL 6347 to (-10, -59.38, -130.88) mm, rotated rx 105.8 ry 33.04 rz 34.05 deg; joints [-5.212, -28.737, 101.579, 146.022, 84.664, 18.837, -475]
  MoveL 6348 to (-8.05, -59.28, -130.75) mm, rotated rx 105.8 ry 33.04 rz 34.05 deg; joints [-5.207, -28.833, 101.764, 146.031, 84.736, 18.787, -475]
  MoveL 6349 to (-6, -59.18, -130.7) mm, rotated rx 105.8 ry 33.04 rz 34.05 deg; joints [-5.206, -28.935, 101.959, 146.037, 84.813, 18.734, -475]
  MoveL 6350 to (-3.87, -59.06, -130.68) mm, rotated rx 105.8 ry 33.04 rz 34.05 deg; joints [-5.205, -29.04, 102.16, 146.042, 84.893, 18.68, -475]
  MoveL 6351 to (-1.75, -58.95, -130.56) mm, rotated rx 105.8 ry 33.04 rz 34.05 deg; joints [-5.201, -29.144, 102.361, 146.051, 84.972, 18.625, -475]
  MoveL 6352 to (0.53, -58.83, -130.3) mm, rotated rx 105.8 ry 33.04 rz 34.05 deg; joints [-5.192, -29.257, 102.576, 146.065, 85.056, 18.565, -475]
  MoveL 6353 to (2.93, -58.7, -130.11) mm, rotated rx 105.8 ry 33.04 rz 34.05 deg; joints [-5.185, -29.374, 102.802, 146.077, 85.145, 18.503, -475]
  MoveL 6354 to (5.26, -58.57, -129.91) mm, rotated rx 105.8 ry 33.04 rz 34.05 deg; joints [-5.178, -29.488, 103.021, 146.089, 85.231, 18.442, -475]
  MoveL 6355 to (7.39, -58.44, -129.8) mm, rotated rx 105.8 ry 33.04 rz 34.05 deg; joints [-5.174, -29.592, 103.221, 146.097, 85.31, 18.388, -475]
  MoveL 6356 to (11.61, -58.19, -129.52) mm, rotated rx 105.8 ry 33.04 rz 34.05 deg; joints [-5.165, -29.797, 103.616, 146.115, 85.467, 18.279, -475]
  MoveL 6357 to (13.78, -58.06, -129.46) mm, rotated rx 105.8 ry 33.04 rz 34.05 deg; joints [-5.163, -29.902, 103.819, 146.121, 85.547, 18.224, -475]
  MoveL 6358 to (15.91, -57.92, -129.24) mm, rotated rx 105.8 ry 33.04 rz 34.05 deg; joints [-5.154, -30.004, 104.017, 146.133, 85.626, 18.168, -475]
  MoveL 6359 to (18.01, -57.77, -129.08) mm, rotated rx 105.8 ry 33.04 rz 34.05 deg; joints [-5.149, -30.105, 104.214, 146.143, 85.704, 18.114, -475]
  MoveL 6360 to (20.12, -57.62, -128.89) mm, rotated rx 105.8 ry 33.04 rz 34.05 deg; joints [-5.142, -30.206, 104.41, 146.153, 85.783, 18.059, -475]
  MoveL 6361 to (22.29, -57.49, -128.8) mm, rotated rx 105.8 ry 33.04 rz 34.05 deg; joints [-5.139, -30.31, 104.611, 146.16, 85.863, 18.004, -475]
  MoveL 6362 to (24.56, -57.32, -128.67) mm, rotated rx 105.8 ry 33.04 rz 34.05 deg; joints [-5.134, -30.418, 104.822, 146.169, 85.948, 17.945, -475]
  MoveL 6363 to (26.46, -57.22, -128.61) mm, rotated rx 105.8 ry 33.04 rz 34.05 deg; joints [-5.132, -30.51, 104.998, 146.174, 86.017, 17.898, -475]
  MoveL 6364 to (26.42, -56.56, -127.73) mm, rotated rx 105.8 ry 33.04 rz 34.05 deg; joints [-5.098, -30.478, 105.002, 146.209, 86.042, 17.87, -475]
  MoveL 6365 to (26.12, -56.36, -127.32) mm, rotated rx 105.8 ry 33.04 rz 34.05 deg; joints [-5.081, -30.454, 104.977, 146.226, 86.038, 17.867, -475]
  MoveL 6366 to (26.09, -56.3, -127.04) mm, rotated rx 105.8 ry 33.04 rz 34.05 deg; joints [-5.07, -30.449, 104.975, 146.236, 86.039, 17.863, -475]
  MoveL 6367 to (26.4, -56.42, -126.92) mm, rotated rx 105.8 ry 33.04 rz 34.05 deg; joints [-5.066, -30.47, 105.002, 146.241, 86.043, 17.859, -475]
  MoveL 6368 to (26.8, -56.62, -126.86) mm, rotated rx 105.8 ry 33.04 rz 34.05 deg; joints [-5.063, -30.5, 105.037, 146.244, 86.048, 17.855, -475]
  MoveL 6369 to (27.3, -56.88, -126.83) mm, rotated rx 105.8 ry 33.04 rz 34.05 deg; joints [-5.062, -30.537, 105.08, 146.245, 86.052, 17.852, -475]
  MoveL 6370 to (27.91, -57.21, -126.79) mm, rotated rx 105.8 ry 33.04 rz 34.05 deg; joints [-5.06, -30.582, 105.132, 146.247, 86.057, 17.848, -475]
  MoveL 6371 to (28.46, -57.53, -126.76) mm, rotated rx 105.8 ry 33.04 rz 34.05 deg; joints [-5.059, -30.624, 105.179, 146.248, 86.062, 17.845, -475]
  MoveL 6372 to (28.91, -57.79, -126.76) mm, rotated rx 105.8 ry 33.04 rz 34.05 deg; joints [-5.059, -30.659, 105.218, 146.249, 86.065, 17.843, -475]
  MoveL 6373 to (29.34, -58.03, -126.75) mm, rotated rx 105.8 ry 33.04 rz 34.05 deg; joints [-5.058, -30.691, 105.254, 146.249, 86.068, 17.84, -475]
  MoveL 6374 to (30.26, -58.51, -126.67) mm, rotated rx 105.8 ry 33.04 rz 34.05 deg; joints [-5.055, -30.76, 105.333, 146.253, 86.076, 17.833, -475]
  MoveL 6375 to (30.76, -58.77, -126.62) mm, rotated rx 105.8 ry 33.04 rz 34.05 deg; joints [-5.053, -30.797, 105.376, 146.255, 86.081, 17.83, -475]
  MoveL 6376 to (31.22, -58.99, -126.55) mm, rotated rx 105.8 ry 33.04 rz 34.05 deg; joints [-5.05, -30.83, 105.416, 146.258, 86.086, 17.825, -475]
  MoveL 6377 to (31.64, -59.18, -126.48) mm, rotated rx 105.8 ry 33.04 rz 34.05 deg; joints [-5.047, -30.86, 105.452, 146.261, 86.091, 17.821, -475]
  MoveL 6378 to (32.06, -59.39, -126.42) mm, rotated rx 105.8 ry 33.04 rz 34.05 deg; joints [-5.045, -30.89, 105.488, 146.264, 86.096, 17.817, -475]
  MoveL 6379 to (32.48, -59.61, -126.39) mm, rotated rx 105.8 ry 33.04 rz 34.05 deg; joints [-5.044, -30.922, 105.525, 146.265, 86.099, 17.814, -475]
  MoveL 6380 to (32.94, -59.87, -126.37) mm, rotated rx 105.8 ry 33.04 rz 34.05 deg; joints [-5.043, -30.956, 105.564, 146.266, 86.103, 17.812, -475]
  MoveL 6381 to (36.09, -61.74, -126.37) mm, rotated rx 105.8 ry 33.04 rz 34.05 deg; joints [-5.042, -31.2, 105.831, 146.268, 86.122, 17.799, -475]
  MoveL 6382 to (37.43, -62.66, -126.39) mm, rotated rx 105.8 ry 33.04 rz 34.05 deg; joints [-5.043, -31.31, 105.942, 146.267, 86.124, 17.798, -475]
  MoveL 6383 to (37.85, -63.06, -126.42) mm, rotated rx 105.8 ry 33.04 rz 34.05 deg; joints [-5.044, -31.349, 105.976, 146.266, 86.12, 17.801, -475]
  MoveL 6384 to (38.11, -63.42, -126.45) mm, rotated rx 105.8 ry 33.04 rz 34.05 deg; joints [-5.045, -31.378, 105.995, 146.264, 86.112, 17.807, -475]
  MoveL 6385 to (38.23, -63.73, -126.49) mm, rotated rx 105.8 ry 33.04 rz 34.05 deg; joints [-5.047, -31.398, 106.003, 146.262, 86.101, 17.814, -475]
  MoveL 6386 to (38.24, -63.88, -126.52) mm, rotated rx 105.8 ry 33.04 rz 34.05 deg; joints [-5.048, -31.406, 106.002, 146.261, 86.095, 17.819, -475]
  MoveL 6387 to (38.22, -64.02, -126.54) mm, rotated rx 105.8 ry 33.04 rz 34.05 deg; joints [-5.048, -31.411, 105.999, 146.26, 86.088, 17.824, -475]
  MoveL 6388 to (38.17, -64.15, -126.57) mm, rotated rx 105.8 ry 33.04 rz 34.05 deg; joints [-5.049, -31.414, 105.993, 146.259, 86.08, 17.829, -475]
  MoveL 6389 to (38.1, -64.27, -126.6) mm, rotated rx 105.8 ry 33.04 rz 34.05 deg; joints [-5.051, -31.416, 105.985, 146.257, 86.072, 17.835, -475]
  MoveL 6390 to (37.87, -64.49, -126.66) mm, rotated rx 105.8 ry 33.04 rz 34.05 deg; joints [-5.053, -31.414, 105.962, 146.254, 86.055, 17.847, -475]
  MoveL 6391 to (37.16, -64.85, -126.79) mm, rotated rx 105.8 ry 33.04 rz 34.05 deg; joints [-5.058, -31.394, 105.893, 146.248, 86.015, 17.876, -475]
  MoveL 6392 to (36.19, -65.11, -126.93) mm, rotated rx 105.8 ry 33.04 rz 34.05 deg; joints [-5.063, -31.357, 105.801, 146.24, 85.971, 17.907, -475]
  MoveL 6393 to (33.87, -65.41, -127.2) mm, rotated rx 105.8 ry 33.04 rz 34.05 deg; joints [-5.073, -31.252, 105.586, 146.226, 85.88, 17.971, -475]
  MoveL 6394 to (31.46, -65.57, -127.44) mm, rotated rx 105.8 ry 33.04 rz 34.05 deg; joints [-5.082, -31.137, 105.364, 146.213, 85.793, 18.032, -475]
  MoveL 6395 to (-22.43, -68.71, -132.52) mm, rotated rx 105.8 ry 33.04 rz 34.05 deg; joints [-5.266, -28.487, 100.293, 145.91, 83.814, 19.434, -475]
  MoveL 6396 to (-26.26, -68.94, -132.88) mm, rotated rx 105.8 ry 33.04 rz 34.05 deg; joints [-5.279, -28.295, 99.925, 145.887, 83.67, 19.537, -475]
  MoveL 6397 to (-30.01, -68.97, -133.3) mm, rotated rx 105.8 ry 33.04 rz 34.05 deg; joints [-5.294, -28.099, 99.565, 145.862, 83.537, 19.633, -475]
  MoveL 6398 to (-31.47, -68.71, -133.51) mm, rotated rx 105.8 ry 33.04 rz 34.05 deg; joints [-5.301, -28.01, 99.426, 145.851, 83.497, 19.664, -475]
  MoveL 6399 to (-31.97, -68.47, -133.6) mm, rotated rx 105.8 ry 33.04 rz 34.05 deg; joints [-5.305, -27.974, 99.382, 145.847, 83.491, 19.67, -475]
  MoveL 6400 to (-32.13, -68.32, -133.65) mm, rotated rx 105.8 ry 33.04 rz 34.05 deg; joints [-5.307, -27.959, 99.368, 145.845, 83.492, 19.67, -475]
  MoveL 6401 to (-32.24, -68.14, -133.69) mm, rotated rx 105.8 ry 33.04 rz 34.05 deg; joints [-5.308, -27.946, 99.359, 145.844, 83.496, 19.667, -475]
  MoveL 6402 to (-32.29, -67.94, -133.73) mm, rotated rx 105.8 ry 33.04 rz 34.05 deg; joints [-5.31, -27.935, 99.357, 145.843, 83.504, 19.663, -475]
  MoveL 6403 to (-32.26, -67.71, -133.76) mm, rotated rx 105.8 ry 33.04 rz 34.05 deg; joints [-5.311, -27.927, 99.362, 145.843, 83.515, 19.655, -475]
  MoveL 6404 to (-32.16, -67.45, -133.79) mm, rotated rx 105.8 ry 33.04 rz 34.05 deg; joints [-5.313, -27.921, 99.375, 145.842, 83.53, 19.646, -475]
  MoveL 6405 to (-31.99, -67.16, -133.82) mm, rotated rx 105.8 ry 33.04 rz 34.05 deg; joints [-5.314, -27.918, 99.395, 145.843, 83.55, 19.633, -475]
  MoveL 6406 to (-30.39, -65.66, -133.87) mm, rotated rx 105.8 ry 33.04 rz 34.05 deg; joints [-5.317, -27.939, 99.566, 145.849, 83.674, 19.549, -475]
  MoveL 6407 to (-28.72, -64.39, -133.87) mm, rotated rx 105.8 ry 33.04 rz 34.05 deg; joints [-5.318, -27.974, 99.74, 145.856, 83.79, 19.471, -475]
  MoveL 6408 to (-25.42, -62.49, -133.91) mm, rotated rx 105.8 ry 33.04 rz 34.05 deg; joints [-5.322, -28.067, 100.077, 145.867, 83.993, 19.334, -475]
  MoveL 6409 to (-22.04, -61.43, -134.02) mm, rotated rx 105.8 ry 33.04 rz 34.05 deg; joints [-5.328, -28.199, 100.412, 145.873, 84.162, 19.221, -475]
  MoveL 6410 to (-16, -61.08, -134.32) mm, rotated rx 105.8 ry 33.04 rz 34.05 deg; joints [-5.342, -28.499, 100.99, 145.875, 84.394, 19.068, -475]
  MoveL 6411 to (-13.67, -61.43, -134.45) mm, rotated rx 105.8 ry 33.04 rz 34.05 deg; joints [-5.347, -28.636, 101.207, 145.874, 84.462, 19.024, -475]
  MoveL 6412 to (20.45, -68.13, -136.31) mm, rotated rx 105.8 ry 33.04 rz 34.05 deg; joints [-5.429, -30.689, 104.317, 145.847, 85.349, 18.449, -475]
  MoveL 6413 to (23.37, -68.69, -136.48) mm, rotated rx 105.8 ry 33.04 rz 34.05 deg; joints [-5.436, -30.864, 104.578, 145.844, 85.422, 18.401, -475]
  MoveL 6414 to (27.1, -68.94, -136.72) mm, rotated rx 105.8 ry 33.04 rz 34.05 deg; joints [-5.447, -31.066, 104.918, 145.839, 85.537, 18.326, -475]
  MoveL 6415 to (28.56, -68.71, -136.86) mm, rotated rx 105.8 ry 33.04 rz 34.05 deg; joints [-5.454, -31.131, 105.054, 145.836, 85.598, 18.287, -475]
  MoveL 6416 to (29.05, -68.47, -136.93) mm, rotated rx 105.8 ry 33.04 rz 34.05 deg; joints [-5.457, -31.145, 105.102, 145.835, 85.626, 18.269, -475]
  MoveL 6417 to (29.22, -68.32, -136.96) mm, rotated rx 105.8 ry 33.04 rz 34.05 deg; joints [-5.459, -31.147, 105.119, 145.834, 85.639, 18.261, -475]
  MoveL 6418 to (29.33, -68.14, -137) mm, rotated rx 105.8 ry 33.04 rz 34.05 deg; joints [-5.46, -31.144, 105.131, 145.833, 85.651, 18.253, -475]
  MoveL 6419 to (29.37, -67.93, -137.03) mm, rotated rx 105.8 ry 33.04 rz 34.05 deg; joints [-5.462, -31.137, 105.137, 145.832, 85.662, 18.246, -475]
  MoveL 6420 to (29.34, -67.7, -137.07) mm, rotated rx 105.8 ry 33.04 rz 34.05 deg; joints [-5.463, -31.126, 105.137, 145.831, 85.672, 18.24, -475]
  MoveL 6421 to (29.24, -67.44, -137.1) mm, rotated rx 105.8 ry 33.04 rz 34.05 deg; joints [-5.465, -31.109, 105.131, 145.83, 85.681, 18.234, -475]
  MoveL 6422 to (29.06, -67.14, -137.14) mm, rotated rx 105.8 ry 33.04 rz 34.05 deg; joints [-5.466, -31.087, 105.118, 145.829, 85.689, 18.23, -475]
  MoveL 6423 to (27.45, -65.66, -137.26) mm, rotated rx 105.8 ry 33.04 rz 34.05 deg; joints [-5.471, -30.939, 104.987, 145.825, 85.704, 18.221, -475]
  MoveL 6424 to (27.03, -65.35, -137.28) mm, rotated rx 105.8 ry 33.04 rz 34.05 deg; joints [-5.472, -30.904, 104.952, 145.824, 85.704, 18.221, -475]
  MoveL 6425 to (26.65, -65.1, -137.33) mm, rotated rx 105.8 ry 33.04 rz 34.05 deg; joints [-5.474, -30.873, 104.92, 145.822, 85.703, 18.222, -475]
  MoveL 6426 to (26.27, -64.88, -137.4) mm, rotated rx 105.8 ry 33.04 rz 34.05 deg; joints [-5.477, -30.843, 104.888, 145.819, 85.701, 18.225, -475]
  MoveL 6427 to (25.9, -64.64, -137.46) mm, rotated rx 105.8 ry 33.04 rz 34.05 deg; joints [-5.479, -30.814, 104.856, 145.817, 85.7, 18.226, -475]
  MoveL 6428 to (25.51, -64.37, -137.49) mm, rotated rx 105.8 ry 33.04 rz 34.05 deg; joints [-5.48, -30.783, 104.824, 145.815, 85.699, 18.227, -475]
  MoveL 6429 to (21.81, -61.5, -137.5) mm, rotated rx 105.8 ry 33.04 rz 34.05 deg; joints [-5.481, -30.466, 104.516, 145.815, 85.706, 18.223, -475]
  MoveL 6430 to (21.46, -61.24, -137.52) mm, rotated rx 105.8 ry 33.04 rz 34.05 deg; joints [-5.482, -30.437, 104.486, 145.814, 85.706, 18.223, -475]
  MoveL 6431 to (21.08, -60.95, -137.53) mm, rotated rx 105.8 ry 33.04 rz 34.05 deg; joints [-5.482, -30.404, 104.454, 145.814, 85.707, 18.223, -475]
  MoveL 6432 to (20.26, -60.32, -137.53) mm, rotated rx 105.8 ry 33.04 rz 34.05 deg; joints [-5.482, -30.335, 104.386, 145.814, 85.708, 18.222, -475]
  MoveL 6433 to (19.8, -59.97, -137.54) mm, rotated rx 105.8 ry 33.04 rz 34.05 deg; joints [-5.483, -30.296, 104.347, 145.814, 85.708, 18.222, -475]
  MoveL 6434 to (19.31, -59.63, -137.56) mm, rotated rx 105.8 ry 33.04 rz 34.05 deg; joints [-5.483, -30.255, 104.305, 145.813, 85.707, 18.223, -475]
  MoveL 6435 to (18.74, -59.28, -137.59) mm, rotated rx 105.8 ry 33.04 rz 34.05 deg; joints [-5.484, -30.211, 104.257, 145.812, 85.704, 18.226, -475]
  MoveL 6436 to (18.14, -59, -137.61) mm, rotated rx 105.8 ry 33.04 rz 34.05 deg; joints [-5.485, -30.168, 104.204, 145.81, 85.696, 18.231, -475]
  MoveL 6437 to (17.53, -58.78, -137.63) mm, rotated rx 105.8 ry 33.04 rz 34.05 deg; joints [-5.486, -30.127, 104.15, 145.809, 85.685, 18.238, -475]
  MoveL 6438 to (18.63, -59.49, -138.61) mm, rotated rx 105.8 ry 33.04 rz 34.05 deg; joints [-5.524, -30.215, 104.243, 145.772, 85.695, 18.245, -475]
  MoveL 6439 to (17.31, -59.72, -139.03) mm, rotated rx 105.8 ry 33.04 rz 34.05 deg; joints [-5.541, -30.158, 104.118, 145.753, 85.642, 18.287, -475]
  MoveL 6440 to (15.82, -59.83, -139.35) mm, rotated rx 105.8 ry 33.04 rz 34.05 deg; joints [-5.552, -30.087, 103.979, 145.738, 85.587, 18.328, -475]
  MoveL 6441 to (14.12, -59.85, -139.59) mm, rotated rx 105.8 ry 33.04 rz 34.05 deg; joints [-5.561, -30.001, 103.821, 145.727, 85.529, 18.37, -475]
  MoveL 6442 to (11.99, -59.75, -139.81) mm, rotated rx 105.8 ry 33.04 rz 34.05 deg; joints [-5.568, -29.887, 103.624, 145.716, 85.462, 18.419, -475]
  MoveL 6443 to (9.86, -59.62, -139.92) mm, rotated rx 105.8 ry 33.04 rz 34.05 deg; joints [-5.572, -29.772, 103.428, 145.709, 85.395, 18.466, -475]
  MoveL 6444 to (7.73, -59.49, -140.03) mm, rotated rx 105.8 ry 33.04 rz 34.05 deg; joints [-5.575, -29.657, 103.231, 145.702, 85.328, 18.513, -475]
  MoveL 6445 to (5.6, -59.37, -140.26) mm, rotated rx 105.8 ry 33.04 rz 34.05 deg; joints [-5.583, -29.543, 103.033, 145.69, 85.261, 18.562, -475]
  MoveL 6446 to (3.47, -59.23, -140.38) mm, rotated rx 105.8 ry 33.04 rz 34.05 deg; joints [-5.587, -29.427, 102.836, 145.683, 85.193, 18.609, -475]
  MoveL 6447 to (1.34, -59.1, -140.61) mm, rotated rx 105.8 ry 33.04 rz 34.05 deg; joints [-5.595, -29.312, 102.638, 145.671, 85.126, 18.658, -475]
  MoveL 6448 to (-0.79, -58.95, -140.73) mm, rotated rx 105.8 ry 33.04 rz 34.05 deg; joints [-5.599, -29.196, 102.44, 145.663, 85.059, 18.705, -475]
  MoveL 6449 to (-2.92, -58.81, -140.84) mm, rotated rx 105.8 ry 33.04 rz 34.05 deg; joints [-5.602, -29.08, 102.242, 145.656, 84.992, 18.752, -475]
  MoveL 6450 to (-5.05, -58.66, -141.08) mm, rotated rx 105.8 ry 33.04 rz 34.05 deg; joints [-5.61, -28.964, 102.043, 145.644, 84.925, 18.801, -475]
  MoveL 6451 to (-7.08, -58.5, -141.18) mm, rotated rx 105.8 ry 33.04 rz 34.05 deg; joints [-5.614, -28.852, 101.853, 145.637, 84.861, 18.846, -475]
  MoveL 6452 to (-9.06, -58.35, -141.39) mm, rotated rx 105.8 ry 33.04 rz 34.05 deg; joints [-5.621, -28.743, 101.668, 145.626, 84.8, 18.891, -475]
  MoveL 6453 to (-11.43, -58.19, -141.55) mm, rotated rx 105.8 ry 33.04 rz 34.05 deg; joints [-5.626, -28.613, 101.446, 145.616, 84.724, 18.945, -475]
  MoveL 6454 to (-14.14, -57.96, -141.64) mm, rotated rx 105.8 ry 33.04 rz 34.05 deg; joints [-5.628, -28.463, 101.191, 145.609, 84.639, 19.004, -475]
  MoveL 6455 to (-16.21, -57.81, -141.71) mm, rotated rx 105.8 ry 33.04 rz 34.05 deg; joints [-5.629, -28.349, 100.997, 145.603, 84.572, 19.05, -475]
  MoveL 6456 to (-18.13, -57.67, -141.83) mm, rotated rx 105.8 ry 33.04 rz 34.05 deg; joints [-5.634, -28.243, 100.816, 145.595, 84.511, 19.094, -475]
  MoveL 6457 to (-20.11, -57.52, -141.94) mm, rotated rx 105.8 ry 33.04 rz 34.05 deg; joints [-5.637, -28.134, 100.629, 145.587, 84.448, 19.139, -475]
  MoveL 6458 to (-22.05, -57.37, -142.05) mm, rotated rx 105.8 ry 33.04 rz 34.05 deg; joints [-5.64, -28.026, 100.445, 145.58, 84.386, 19.183, -475]
  MoveL 6459 to (-24.11, -57.21, -142.12) mm, rotated rx 105.8 ry 33.04 rz 34.05 deg; joints [-5.642, -27.912, 100.25, 145.574, 84.319, 19.229, -475]
  MoveL 6460 to (-26.32, -57.03, -142.22) mm, rotated rx 105.8 ry 33.04 rz 34.05 deg; joints [-5.644, -27.789, 100.04, 145.566, 84.248, 19.279, -475]
  MoveL 6461 to (-28.72, -56.81, -142.48) mm, rotated rx 105.8 ry 33.04 rz 34.05 deg; joints [-5.653, -27.654, 99.813, 145.552, 84.173, 19.334, -475]
  MoveL 6462 to (-30.94, -57.13, -143.46) mm, rotated rx 105.8 ry 33.04 rz 34.05 deg; joints [-5.69, -27.551, 99.595, 145.51, 84.084, 19.409, -475]
  MoveL 6463 to (-29.94, -56.57, -143.95) mm, rotated rx 105.8 ry 33.04 rz 34.05 deg; joints [-5.709, -27.58, 99.696, 145.495, 84.147, 19.373, -475]
  MoveL 6464 to (-29.42, -56.28, -144.26) mm, rotated rx 105.8 ry 33.04 rz 34.05 deg; joints [-5.722, -27.595, 99.749, 145.485, 84.181, 19.354, -475]
  MoveL 6465 to (-29.34, -56.23, -144.41) mm, rotated rx 105.8 ry 33.04 rz 34.05 deg; joints [-5.728, -27.597, 99.757, 145.48, 84.187, 19.352, -475]
  MoveL 6466 to (-29.64, -56.39, -144.45) mm, rotated rx 105.8 ry 33.04 rz 34.05 deg; joints [-5.729, -27.588, 99.726, 145.477, 84.169, 19.365, -475]
  MoveL 6467 to (-30.05, -56.62, -144.46) mm, rotated rx 105.8 ry 33.04 rz 34.05 deg; joints [-5.729, -27.576, 99.684, 145.475, 84.144, 19.382, -475]
  MoveL 6468 to (-30.47, -56.84, -144.5) mm, rotated rx 105.8 ry 33.04 rz 34.05 deg; joints [-5.73, -27.563, 99.641, 145.473, 84.12, 19.4, -475]
  MoveL 6469 to (-30.88, -57.03, -144.56) mm, rotated rx 105.8 ry 33.04 rz 34.05 deg; joints [-5.732, -27.55, 99.6, 145.469, 84.097, 19.416, -475]
  MoveL 6470 to (-31.29, -57.23, -144.6) mm, rotated rx 105.8 ry 33.04 rz 34.05 deg; joints [-5.733, -27.537, 99.558, 145.466, 84.073, 19.433, -475]
  MoveL 6471 to (-31.73, -57.47, -144.62) mm, rotated rx 105.8 ry 33.04 rz 34.05 deg; joints [-5.733, -27.524, 99.514, 145.464, 84.047, 19.451, -475]
  MoveL 6472 to (-34, -58.77, -144.62) mm, rotated rx 105.8 ry 33.04 rz 34.05 deg; joints [-5.731, -27.46, 99.281, 145.456, 83.908, 19.547, -475]
  MoveL 6473 to (-34.4, -58.98, -144.64) mm, rotated rx 105.8 ry 33.04 rz 34.05 deg; joints [-5.731, -27.448, 99.239, 145.454, 83.884, 19.563, -475]
  MoveL 6474 to (-34.75, -59.15, -144.67) mm, rotated rx 105.8 ry 33.04 rz 34.05 deg; joints [-5.732, -27.437, 99.204, 145.452, 83.864, 19.577, -475]
  MoveL 6475 to (-35.16, -59.37, -144.69) mm, rotated rx 105.8 ry 33.04 rz 34.05 deg; joints [-5.733, -27.424, 99.162, 145.449, 83.84, 19.594, -475]
  MoveL 6476 to (-35.68, -59.65, -144.71) mm, rotated rx 105.8 ry 33.04 rz 34.05 deg; joints [-5.733, -27.409, 99.109, 145.447, 83.809, 19.616, -475]
  MoveL 6477 to (-36.33, -59.98, -144.77) mm, rotated rx 105.8 ry 33.04 rz 34.05 deg; joints [-5.735, -27.388, 99.043, 145.442, 83.772, 19.642, -475]
  MoveL 6478 to (-36.88, -60.27, -144.8) mm, rotated rx 105.8 ry 33.04 rz 34.05 deg; joints [-5.735, -27.372, 98.987, 145.439, 83.739, 19.665, -475]
  MoveL 6479 to (-37.34, -60.53, -144.8) mm, rotated rx 105.8 ry 33.04 rz 34.05 deg; joints [-5.735, -27.358, 98.939, 145.438, 83.711, 19.685, -475]
  MoveL 6480 to (-38.71, -61.31, -144.8) mm, rotated rx 105.8 ry 33.04 rz 34.05 deg; joints [-5.734, -27.319, 98.798, 145.433, 83.627, 19.742, -475]
  MoveL 6481 to (-41.37, -62.49, -145.14) mm, rotated rx 105.8 ry 33.04 rz 34.05 deg; joints [-5.744, -27.228, 98.527, 145.411, 83.481, 19.848, -475]
  MoveL 6482 to (-42.63, -62.79, -145.57) mm, rotated rx 105.8 ry 33.04 rz 34.05 deg; joints [-5.76, -27.173, 98.4, 145.391, 83.425, 19.893, -475]
  MoveL 6483 to (-43.84, -62.89, -146.17) mm, rotated rx 105.8 ry 33.04 rz 34.05 deg; joints [-5.782, -27.113, 98.28, 145.365, 83.379, 19.933, -475]
  MoveL 6484 to (-46.13, -62.5, -147.88) mm, rotated rx 105.8 ry 33.04 rz 34.05 deg; joints [-5.845, -26.975, 98.059, 145.298, 83.322, 19.998, -475]
  MoveL 6485 to (-48.23, -61.33, -150.28) mm, rotated rx 105.8 ry 33.04 rz 34.05 deg; joints [-5.936, -26.814, 97.863, 145.207, 83.31, 20.043, -475]
  MoveL 6486 to (-49.62, -59.81, -152.67) mm, rotated rx 105.8 ry 33.04 rz 34.05 deg; joints [-6.026, -26.677, 97.739, 145.119, 83.338, 20.059, -475]
  MoveL 6487 to (-49.86, -59.08, -153.61) mm, rotated rx 105.8 ry 33.04 rz 34.05 deg; joints [-6.062, -26.634, 97.722, 145.086, 83.366, 20.054, -475]
  MoveL 6488 to (-49.78, -58.38, -154.38) mm, rotated rx 105.8 ry 33.04 rz 34.05 deg; joints [-6.092, -26.609, 97.735, 145.059, 83.403, 20.039, -475]
  MoveL 6489 to (-49.62, -58.03, -154.7) mm, rotated rx 105.8 ry 33.04 rz 34.05 deg; joints [-6.105, -26.602, 97.754, 145.049, 83.425, 20.029, -475]
  MoveL 6490 to (-49.39, -57.69, -154.98) mm, rotated rx 105.8 ry 33.04 rz 34.05 deg; joints [-6.116, -26.601, 97.779, 145.04, 83.45, 20.016, -475]
  MoveL 6491 to (-48.7, -57.03, -155.41) mm, rotated rx 105.8 ry 33.04 rz 34.05 deg; joints [-6.133, -26.61, 97.853, 145.027, 83.506, 19.983, -475]
  MoveL 6492 to (-47.69, -56.39, -155.67) mm, rotated rx 105.8 ry 33.04 rz 34.05 deg; joints [-6.144, -26.636, 97.957, 145.021, 83.572, 19.941, -475]
  MoveL 6493 to (-46.38, -55.78, -155.75) mm, rotated rx 105.8 ry 33.04 rz 34.05 deg; joints [-6.149, -26.68, 98.092, 145.022, 83.647, 19.89, -475]
  MoveL 6494 to (-45.89, -55.58, -155.75) mm, rotated rx 105.8 ry 33.04 rz 34.05 deg; joints [-6.149, -26.697, 98.141, 145.024, 83.673, 19.872, -475]
  MoveL 6495 to (-45.48, -55.45, -155.7) mm, rotated rx 105.8 ry 33.04 rz 34.05 deg; joints [-6.148, -26.714, 98.183, 145.027, 83.694, 19.856, -475]
  MoveL 6496 to (-45.06, -55.32, -155.64) mm, rotated rx 105.8 ry 33.04 rz 34.05 deg; joints [-6.146, -26.73, 98.225, 145.031, 83.715, 19.841, -475]
  MoveL 6497 to (-44.61, -55.16, -155.6) mm, rotated rx 105.8 ry 33.04 rz 34.05 deg; joints [-6.145, -26.747, 98.27, 145.033, 83.738, 19.825, -475]
  MoveL 6498 to (-44.15, -54.99, -155.58) mm, rotated rx 105.8 ry 33.04 rz 34.05 deg; joints [-6.145, -26.764, 98.317, 145.035, 83.762, 19.808, -475]
  MoveL 6499 to (-43.65, -54.79, -155.58) mm, rotated rx 105.8 ry 33.04 rz 34.05 deg; joints [-6.145, -26.782, 98.368, 145.037, 83.789, 19.789, -475]
  MoveL 6500 to (-43.17, -54.59, -155.58) mm, rotated rx 105.8 ry 33.04 rz 34.05 deg; joints [-6.146, -26.799, 98.417, 145.038, 83.815, 19.771, -475]
  MoveL 6501 to (-42.71, -54.38, -155.59) mm, rotated rx 105.8 ry 33.04 rz 34.05 deg; joints [-6.147, -26.815, 98.464, 145.039, 83.841, 19.753, -475]
  MoveL 6502 to (-42.25, -54.18, -155.6) mm, rotated rx 105.8 ry 33.04 rz 34.05 deg; joints [-6.148, -26.831, 98.51, 145.04, 83.866, 19.736, -475]
  MoveL 6503 to (-41.82, -54.02, -155.58) mm, rotated rx 105.8 ry 33.04 rz 34.05 deg; joints [-6.148, -26.847, 98.554, 145.042, 83.889, 19.719, -475]
  MoveL 6504 to (-41.38, -53.86, -155.54) mm, rotated rx 105.8 ry 33.04 rz 34.05 deg; joints [-6.146, -26.863, 98.598, 145.045, 83.911, 19.703, -475]
  MoveL 6505 to (-40.87, -53.69, -155.49) mm, rotated rx 105.8 ry 33.04 rz 34.05 deg; joints [-6.145, -26.883, 98.65, 145.048, 83.938, 19.684, -475]
  MoveL 6506 to (-40.2, -53.46, -155.44) mm, rotated rx 105.8 ry 33.04 rz 34.05 deg; joints [-6.144, -26.908, 98.717, 145.052, 83.971, 19.66, -475]
  MoveL 6507 to (-39.6, -53.23, -155.42) mm, rotated rx 105.8 ry 33.04 rz 34.05 deg; joints [-6.144, -26.93, 98.778, 145.055, 84.003, 19.638, -475]
  MoveL 6508 to (-37.18, -52.23, -155.42) mm, rotated rx 105.8 ry 33.04 rz 34.05 deg; joints [-6.146, -27.015, 99.022, 145.061, 84.135, 19.546, -475]
  MoveL 6509 to (-36.59, -52.01, -155.38) mm, rotated rx 105.8 ry 33.04 rz 34.05 deg; joints [-6.146, -27.036, 99.081, 145.064, 84.165, 19.525, -475]
  MoveL 6510 to (-36.07, -51.82, -155.32) mm, rotated rx 105.8 ry 33.04 rz 34.05 deg; joints [-6.144, -27.056, 99.134, 145.068, 84.192, 19.505, -475]
  MoveL 6511 to (-35.87, -51.76, -155.17) mm, rotated rx 105.8 ry 33.04 rz 34.05 deg; joints [-6.139, -27.064, 99.154, 145.074, 84.201, 19.497, -475]
  MoveL 6512 to (-35.98, -51.8, -154.91) mm, rotated rx 105.8 ry 33.04 rz 34.05 deg; joints [-6.128, -27.059, 99.143, 145.083, 84.194, 19.498, -475]
  MoveL 6513 to (-36.42, -51.94, -154.5) mm, rotated rx 105.8 ry 33.04 rz 34.05 deg; joints [-6.112, -27.043, 99.101, 145.098, 84.17, 19.509, -475]
  MoveL 6514 to (-35.75, -52.72, -153.7) mm, rotated rx 105.8 ry 33.04 rz 34.05 deg; joints [-6.082, -27.111, 99.159, 145.127, 84.156, 19.507, -475]
  MoveL 6515 to (-33.82, -53.17, -153.48) mm, rotated rx 105.8 ry 33.04 rz 34.05 deg; joints [-6.074, -27.231, 99.341, 145.138, 84.206, 19.469, -475]
  MoveL 6516 to (-31.86, -53.6, -153.32) mm, rotated rx 105.8 ry 33.04 rz 34.05 deg; joints [-6.07, -27.352, 99.525, 145.146, 84.257, 19.431, -475]
  MoveL 6517 to (-29.85, -54.03, -153.17) mm, rotated rx 105.8 ry 33.04 rz 34.05 deg; joints [-6.065, -27.476, 99.714, 145.154, 84.31, 19.393, -475]
  MoveL 6518 to (-28.02, -54.44, -152.88) mm, rotated rx 105.8 ry 33.04 rz 34.05 deg; joints [-6.055, -27.589, 99.886, 145.167, 84.357, 19.356, -475]
  MoveL 6519 to (-25.95, -54.89, -152.69) mm, rotated rx 105.8 ry 33.04 rz 34.05 deg; joints [-6.049, -27.715, 100.08, 145.177, 84.411, 19.316, -475]
  MoveL 6520 to (-23.79, -55.35, -152.51) mm, rotated rx 105.8 ry 33.04 rz 34.05 deg; joints [-6.043, -27.848, 100.282, 145.187, 84.467, 19.275, -475]
  MoveL 6521 to (-21.59, -55.81, -152.42) mm, rotated rx 105.8 ry 33.04 rz 34.05 deg; joints [-6.041, -27.982, 100.487, 145.192, 84.525, 19.234, -475]
  MoveL 6522 to (-18.92, -56.36, -152.33) mm, rotated rx 105.8 ry 33.04 rz 34.05 deg; joints [-6.039, -28.145, 100.736, 145.199, 84.595, 19.184, -475]
  MoveL 6523 to (-17, -56.75, -152.22) mm, rotated rx 105.8 ry 33.04 rz 34.05 deg; joints [-6.036, -28.261, 100.914, 145.205, 84.645, 19.148, -475]
  MoveL 6524 to (-15.21, -57.11, -152.01) mm, rotated rx 105.8 ry 33.04 rz 34.05 deg; joints [-6.029, -28.37, 101.081, 145.215, 84.692, 19.113, -475]
  MoveL 6525 to (-13.23, -57.51, -151.82) mm, rotated rx 105.8 ry 33.04 rz 34.05 deg; joints [-6.023, -28.49, 101.264, 145.225, 84.743, 19.075, -475]
  MoveL 6526 to (-11.14, -57.93, -151.7) mm, rotated rx 105.8 ry 33.04 rz 34.05 deg; joints [-6.02, -28.616, 101.458, 145.231, 84.797, 19.036, -475]
  MoveL 6527 to (-9.06, -58.34, -151.52) mm, rotated rx 105.8 ry 33.04 rz 34.05 deg; joints [-6.014, -28.741, 101.65, 145.24, 84.851, 18.996, -475]
  MoveL 6528 to (-6.99, -58.75, -151.4) mm, rotated rx 105.8 ry 33.04 rz 34.05 deg; joints [-6.011, -28.866, 101.841, 145.247, 84.905, 18.957, -475]
  MoveL 6529 to (-4.85, -59.17, -151.22) mm, rotated rx 105.8 ry 33.04 rz 34.05 deg; joints [-6.005, -28.995, 102.038, 145.256, 84.961, 18.917, -475]
  MoveL 6530 to (-2.76, -59.57, -151.1) mm, rotated rx 105.8 ry 33.04 rz 34.05 deg; joints [-6.002, -29.121, 102.231, 145.263, 85.015, 18.878, -475]
  MoveL 6531 to (-0.66, -59.96, -150.87) mm, rotated rx 105.8 ry 33.04 rz 34.05 deg; joints [-5.994, -29.246, 102.424, 145.274, 85.069, 18.837, -475]
  MoveL 6532 to (1.44, -60.37, -150.76) mm, rotated rx 105.8 ry 33.04 rz 34.05 deg; joints [-5.991, -29.372, 102.616, 145.28, 85.124, 18.798, -475]
  MoveL 6533 to (3.54, -60.76, -150.64) mm, rotated rx 105.8 ry 33.04 rz 34.05 deg; joints [-5.987, -29.497, 102.808, 145.286, 85.178, 18.76, -475]
  MoveL 6534 to (5.64, -61.14, -150.42) mm, rotated rx 105.8 ry 33.04 rz 34.05 deg; joints [-5.98, -29.622, 103.001, 145.297, 85.232, 18.719, -475]
  MoveL 6535 to (7.56, -61.43, -150.21) mm, rotated rx 105.8 ry 33.04 rz 34.05 deg; joints [-5.973, -29.733, 103.176, 145.306, 85.284, 18.681, -475]
  MoveL 6536 to (9.31, -61.63, -149.92) mm, rotated rx 105.8 ry 33.04 rz 34.05 deg; joints [-5.963, -29.832, 103.337, 145.319, 85.334, 18.643, -475]
  MoveL 6537 to (10.93, -61.74, -149.52) mm, rotated rx 105.8 ry 33.04 rz 34.05 deg; joints [-5.948, -29.92, 103.488, 145.337, 85.383, 18.604, -475]
  MoveL 6538 to (9.67, -60.96, -148.59) mm, rotated rx 105.8 ry 33.04 rz 34.05 deg; joints [-5.911, -29.821, 103.381, 145.372, 85.37, 18.599, -475]
  MoveL 6539 to (10.2, -61.18, -148.58) mm, rotated rx 105.8 ry 33.04 rz 34.05 deg; joints [-5.911, -29.858, 103.428, 145.373, 85.378, 18.594, -475]
  MoveL 6540 to (10.68, -61.42, -148.56) mm, rotated rx 105.8 ry 33.04 rz 34.05 deg; joints [-5.91, -29.893, 103.469, 145.374, 85.384, 18.59, -475]
  MoveL 6541 to (11.07, -61.68, -148.5) mm, rotated rx 105.8 ry 33.04 rz 34.05 deg; joints [-5.908, -29.925, 103.504, 145.376, 85.386, 18.588, -475]
  MoveL 6542 to (11.44, -61.93, -148.43) mm, rotated rx 105.8 ry 33.04 rz 34.05 deg; joints [-5.906, -29.955, 103.535, 145.379, 85.386, 18.587, -475]
  MoveL 6543 to (11.8, -62.23, -148.38) mm, rotated rx 105.8 ry 33.04 rz 34.05 deg; joints [-5.904, -29.986, 103.565, 145.381, 85.385, 18.587, -475]
  MoveL 6544 to (12.16, -62.56, -148.35) mm, rotated rx 105.8 ry 33.04 rz 34.05 deg; joints [-5.903, -30.019, 103.595, 145.382, 85.382, 18.588, -475]
  MoveL 6545 to (12.54, -62.92, -148.33) mm, rotated rx 105.8 ry 33.04 rz 34.05 deg; joints [-5.902, -30.055, 103.626, 145.382, 85.378, 18.591, -475]
  MoveL 6546 to (12.91, -63.29, -148.33) mm, rotated rx 105.8 ry 33.04 rz 34.05 deg; joints [-5.902, -30.09, 103.656, 145.382, 85.374, 18.594, -475]
  MoveL 6547 to (13.24, -63.62, -148.32) mm, rotated rx 105.8 ry 33.04 rz 34.05 deg; joints [-5.901, -30.121, 103.684, 145.382, 85.371, 18.596, -475]
  MoveL 6548 to (13.56, -63.9, -148.3) mm, rotated rx 105.8 ry 33.04 rz 34.05 deg; joints [-5.9, -30.15, 103.71, 145.383, 85.368, 18.597, -475]
  MoveL 6549 to (13.91, -64.24, -148.28) mm, rotated rx 105.8 ry 33.04 rz 34.05 deg; joints [-5.9, -30.183, 103.738, 145.383, 85.365, 18.599, -475]
  MoveL 6550 to (14.27, -64.61, -148.28) mm, rotated rx 105.8 ry 33.04 rz 34.05 deg; joints [-5.9, -30.218, 103.768, 145.383, 85.36, 18.602, -475]
  MoveL 6551 to (14.71, -65.04, -148.26) mm, rotated rx 105.8 ry 33.04 rz 34.05 deg; joints [-5.899, -30.259, 103.804, 145.384, 85.356, 18.605, -475]
  MoveL 6552 to (15.22, -65.51, -148.22) mm, rotated rx 105.8 ry 33.04 rz 34.05 deg; joints [-5.897, -30.306, 103.845, 145.385, 85.351, 18.608, -475]
  MoveL 6553 to (15.65, -65.94, -148.2) mm, rotated rx 105.8 ry 33.04 rz 34.05 deg; joints [-5.897, -30.347, 103.881, 145.386, 85.346, 18.611, -475]
  MoveL 6554 to (16.12, -66.38, -148.17) mm, rotated rx 105.8 ry 33.04 rz 34.05 deg; joints [-5.896, -30.39, 103.919, 145.386, 85.342, 18.614, -475]
  MoveL 6555 to (16.64, -66.86, -148.13) mm, rotated rx 105.8 ry 33.04 rz 34.05 deg; joints [-5.894, -30.438, 103.962, 145.388, 85.338, 18.616, -475]
  MoveL 6556 to (17.07, -67.27, -148.12) mm, rotated rx 105.8 ry 33.04 rz 34.05 deg; joints [-5.894, -30.478, 103.996, 145.388, 85.333, 18.619, -475]
  MoveL 6557 to (17.45, -67.66, -148.12) mm, rotated rx 105.8 ry 33.04 rz 34.05 deg; joints [-5.893, -30.515, 104.027, 145.388, 85.328, 18.622, -475]
  MoveL 6558 to (18.56, -68.77, -148.12) mm, rotated rx 105.8 ry 33.04 rz 34.05 deg; joints [-5.893, -30.621, 104.117, 145.387, 85.315, 18.632, -475]
  MoveL 6559 to (19.53, -69.85, -148.2) mm, rotated rx 105.8 ry 33.04 rz 34.05 deg; joints [-5.897, -30.718, 104.193, 145.383, 85.298, 18.644, -475]
  MoveL 6560 to (20.21, -70.83, -148.46) mm, rotated rx 105.8 ry 33.04 rz 34.05 deg; joints [-5.906, -30.795, 104.244, 145.372, 85.278, 18.662, -475]
  MoveL 6561 to (20.59, -71.7, -148.88) mm, rotated rx 105.8 ry 33.04 rz 34.05 deg; joints [-5.923, -30.854, 104.268, 145.355, 85.252, 18.685, -475]
  MoveL 6562 to (20.67, -72.11, -149.15) mm, rotated rx 105.8 ry 33.04 rz 34.05 deg; joints [-5.933, -30.875, 104.27, 145.344, 85.238, 18.699, -475]
